LIN {X 0,Y 493.839,Z 352.42,A -85,B 0,C 180,E1 -6409.672,E2 -6409.672} C_VEL
LIN {X 0,Y 494.204,Z 337.139,A -85,B 0,C 180,E1 -6410.171,E2 -6410.171} C_VEL
LIN {X 0,Y 494.44,Z 322.546,A -85,B 0,C 180,E1 -6410.487,E2 -6410.487} C_VEL
LIN {X 0,Y 495.796,Z 177.299,A -85,B 0,C 180,E1 -6412.659,E2 -6412.659} C_VEL
LIN {X 0,Y 492.339,Z 162.269,A -85,B 0,C 180,E1 -6413.065,E2 -6413.065} C_VEL
LIN {X 0,Y 492.169,Z 161.322,A -85,B 0,C 180,E1 -6413.121,E2 -6413.121} C_VEL
LIN {X 0,Y 492.025,Z 155.5,A -85,B 0,C 180,E1 -6413.912,E2 -6413.912} C_VEL
LIN {X 0,Y 488.755,Z 141.231,A -85,B 0,C 180,E1 -6416.241,E2 -6416.241} C_VEL
LIN {X 0,Y 488.72,Z 141.236,A -85,B 0,C 180,E1 -6419.269,E2 -6419.269} C_VEL
LIN {X 0,Y 488.701,Z 141.23,A -85,B 0,C 180,E1 -6422.146,E2 -6422.146} C_VEL
LIN {X 0,Y 488.719,Z 141.234,A -85,B 0,C 180,E1 -6425.113,E2 -6425.113} C_VEL
LIN {X 0,Y 488.676,Z 141.235,A -85,B 0,C 180,E1 -6428.199,E2 -6428.199} C_VEL
LIN {X 0,Y 488.713,Z 141.229,A -85,B 0,C 180,E1 -6431.413,E2 -6431.413} C_VEL
LIN {X 0,Y 488.695,Z 141.23,A -85,B 0,C 180,E1 -6434.023,E2 -6434.023} C_VEL
LIN {X 0,Y 488.702,Z 141.235,A -85,B 0,C 180,E1 -6437.172,E2 -6437.172} C_VEL
LIN {X 0,Y 488.728,Z 141.23,A -85,B 0,C 180,E1 -6439.676,E2 -6439.676} C_VEL
LIN {X 0,Y 488.674,Z 141.234,A -85,B 0,C 180,E1 -6442.276,E2 -6442.276} C_VEL
LIN {X 0,Y 488.72,Z 141.231,A -85,B 0,C 180,E1 -6445.051,E2 -6445.051} C_VEL
LIN {X 0,Y 488.697,Z 141.232,A -85,B 0,C 180,E1 -6448.044,E2 -6448.044} C_VEL
LIN {X 0,Y 488.725,Z 141.225,A -85,B 0,C 180,E1 -6450.73,E2 -6450.73} C_VEL
LIN {X 0,Y 488.747,Z 141.226,A -85,B 0,C 180,E1 -6453.527,E2 -6453.527} C_VEL
LIN {X 0,Y 488.683,Z 141.23,A -85,B 0,C 180,E1 -6456.254,E2 -6456.254} C_VEL
LIN {X 0,Y 488.735,Z 141.229,A -85,B 0,C 180,E1 -6459.175,E2 -6459.175} C_VEL
LIN {X 0,Y 488.748,Z 141.222,A -85,B 0,C 180,E1 -6461.627,E2 -6461.627} C_VEL
LIN {X 0,Y 488.751,Z 141.228,A -85,B 0,C 180,E1 -6464.999,E2 -6464.999} C_VEL
LIN {X 0,Y 488.797,Z 141.216,A -85,B 0,C 180,E1 -6468.387,E2 -6468.387} C_VEL
LIN {X 0,Y 488.807,Z 141.216,A -85,B 0,C 180,E1 -6471.733,E2 -6471.733} C_VEL
LIN {X 0,Y 488.845,Z 141.206,A -85,B 0,C 180,E1 -6474.224,E2 -6474.224} C_VEL
LIN {X 0,Y 488.951,Z 141.2,A -85,B 0,C 180,E1 -6477.528,E2 -6477.528} C_VEL
LIN {X 0,Y 488.957,Z 141.192,A -85,B 0,C 180,E1 -6480,E2 -6480} C_VEL
LIN {X 0,Y 488.951,Z 141.202,A -85,B 0,C 180,E1 -6482.471,E2 -6482.471} C_VEL
LIN {X 0,Y 488.845,Z 141.208,A -85,B 0,C 180,E1 -6485.776,E2 -6485.776} C_VEL
LIN {X 0,Y 488.807,Z 141.215,A -85,B 0,C 180,E1 -6488.266,E2 -6488.266} C_VEL
LIN {X 0,Y 488.797,Z 141.215,A -85,B 0,C 180,E1 -6491.613,E2 -6491.613} C_VEL
LIN {X 0,Y 488.754,Z 141.225,A -85,B 0,C 180,E1 -6495.001,E2 -6495.001} C_VEL
LIN {X 0,Y 488.744,Z 141.224,A -85,B 0,C 180,E1 -6498.442,E2 -6498.442} C_VEL
LIN {X 0,Y 488.702,Z 141.231,A -85,B 0,C 180,E1 -6501.071,E2 -6501.071} C_VEL
LIN {X 0,Y 488.691,Z 141.23,A -85,B 0,C 180,E1 -6503.745,E2 -6503.745} C_VEL
LIN {X 0,Y 488.781,Z 141.222,A -85,B 0,C 180,E1 -6506.944,E2 -6506.944} C_VEL
LIN {X 0,Y 488.7,Z 141.234,A -85,B 0,C 180,E1 -6510.364,E2 -6510.364} C_VEL
LIN {X 0,Y 488.726,Z 141.227,A -85,B 0,C 180,E1 -6513.485,E2 -6513.485} C_VEL
LIN {X 0,Y 488.68,Z 141.24,A -85,B 0,C 180,E1 -6516.357,E2 -6516.357} C_VEL
LIN {X 0,Y 488.692,Z 141.222,A -85,B 0,C 180,E1 -6519.255,E2 -6519.255} C_VEL
LIN {X 0,Y 488.699,Z 141.221,A -85,B 0,C 180,E1 -6521.601,E2 -6521.601} C_VEL
LIN {X 0,Y 488.704,Z 141.232,A -85,B 0,C 180,E1 -6524.802,E2 -6524.802} C_VEL
LIN {X 0,Y 488.724,Z 141.231,A -85,B 0,C 180,E1 -6527.48,E2 -6527.48} C_VEL
LIN {X 0,Y 488.735,Z 141.227,A -85,B 0,C 180,E1 -6530.751,E2 -6530.751} C_VEL
LIN {X 0,Y 488.678,Z 141.236,A -85,B 0,C 180,E1 -6533.87,E2 -6533.87} C_VEL
LIN {X 0,Y 488.735,Z 141.227,A -85,B 0,C 180,E1 -6536.879,E2 -6536.879} C_VEL
LIN {X 0,Y 488.748,Z 141.374,A -85,B 0,C 180,E1 -6537.233,E2 -6537.233} C_VEL
LIN {X 0,Y 495.388,Z 163.433,A -85,B 0,C 180,E1 -6539.928,E2 -6539.928} C_VEL
LIN {X 0,Y 495.755,Z 164.949,A -85,B 0,C 180,E1 -6540.104,E2 -6540.104} C_VEL
LIN {X 0,Y 494.13,Z 196.323,A -85,B 0,C 180,E1 -6543.157,E2 -6543.157} C_VEL
LIN {X 0,Y 492.556,Z 230.849,A -85,B 0,C 180,E1 -6546.453,E2 -6546.453} C_VEL
LIN {X 0,Y 492.243,Z 239.271,A -85,B 0,C 180,E1 -6547.244,E2 -6547.244} C_VEL
LIN {X 0,Y 494.608,Z 258.487,A -85,B 0,C 180,E1 -6547.65,E2 -6547.65} C_VEL
LIN {X 0,Y 493.264,Z 406.875,A -85,B 0,C 180,E1 -6549.87,E2 -6549.87} C_VEL
LIN {X 0,Y 492.832,Z 422.965,A -85,B 0,C 180,E1 -6550.289,E2 -6550.289} C_VEL
LIN {X 0,Y 492.291,Z 437.461,A -85,B 0,C 180,E1 -6550.833,E2 -6550.833} C_VEL
LIN {X 0,Y 491.618,Z 452.169,A -85,B 0,C 180,E1 -6551.563,E2 -6551.563} C_VEL
LIN {X 0,Y 491.046,Z 465.568,A -85,B 0,C 180,E1 -6552.403,E2 -6552.403} C_VEL
LIN {X 0,Y 490.347,Z 479.102,A -85,B 0,C 180,E1 -6553.443,E2 -6553.443} C_VEL
LIN {X 0,Y 489.704,Z 491.563,A -85,B 0,C 180,E1 -6554.604,E2 -6554.604} C_VEL
LIN {X 0,Y 489.214,Z 502.858,A -85,B 0,C 180,E1 -6555.865,E2 -6555.865} C_VEL
LIN {X 0,Y 488.795,Z 513.821,A -85,B 0,C 180,E1 -6557.335,E2 -6557.335} C_VEL
LIN {X 0,Y 488.506,Z 522.941,A -85,B 0,C 180,E1 -6558.802,E2 -6558.802} C_VEL
LIN {X 0,Y 488.294,Z 529.488,A -85,B 0,C 180,E1 -6560.055,E2 -6560.055} C_VEL
LIN {X 0,Y 488.187,Z 536.746,A -85,B 0,C 180,E1 -6561.724,E2 -6561.724} C_VEL
LIN {X 0,Y 488.144,Z 542.565,A -85,B 0,C 180,E1 -6563.423,E2 -6563.423} C_VEL
LIN {X 0,Y 488.156,Z 546.768,A -85,B 0,C 180,E1 -6565.046,E2 -6565.046} C_VEL
LIN {X 0,Y 488.147,Z 549.786,A -85,B 0,C 180,E1 -6566.7,E2 -6566.7} C_VEL
LIN {X 0,Y 488.087,Z 551.58,A -85,B 0,C 180,E1 -6568.351,E2 -6568.351} C_VEL
LIN {X 0,Y 488.175,Z 552.203,A -85,B 0,C 180,E1 -6570.001,E2 -6570.001} C_VEL
LIN {X 0,Y 488.087,Z 551.582,A -85,B 0,C 180,E1 -6571.651,E2 -6571.651} C_VEL
LIN {X 0,Y 488.161,Z 549.786,A -85,B 0,C 180,E1 -6573.302,E2 -6573.302} C_VEL
LIN {X 0,Y 488.157,Z 546.761,A -85,B 0,C 180,E1 -6574.957,E2 -6574.957} C_VEL
LIN {X 0,Y 488.181,Z 542.448,A -85,B 0,C 180,E1 -6576.614,E2 -6576.614} C_VEL
LIN {X 0,Y 488.223,Z 536.742,A -85,B 0,C 180,E1 -6578.278,E2 -6578.278} C_VEL
LIN {X 0,Y 488.322,Z 529.487,A -85,B 0,C 180,E1 -6579.946,E2 -6579.946} C_VEL
LIN {X 0,Y 488.558,Z 521.718,A -85,B 0,C 180,E1 -6581.409,E2 -6581.409} C_VEL
LIN {X 0,Y 488.825,Z 512.358,A -85,B 0,C 180,E1 -6582.877,E2 -6582.877} C_VEL
LIN {X 0,Y 489.235,Z 502.845,A -85,B 0,C 180,E1 -6584.136,E2 -6584.136} C_VEL
LIN {X 0,Y 489.81,Z 490.499,A -85,B 0,C 180,E1 -6585.501,E2 -6585.501} C_VEL
LIN {X 0,Y 490.392,Z 477.894,A -85,B 0,C 180,E1 -6586.657,E2 -6586.657} C_VEL
LIN {X 0,Y 491.072,Z 463.955,A -85,B 0,C 180,E1 -6587.706,E2 -6587.706} C_VEL
LIN {X 0,Y 491.719,Z 450.208,A -85,B 0,C 180,E1 -6588.544,E2 -6588.544} C_VEL
LIN {X 0,Y 492.335,Z 436.099,A -85,B 0,C 180,E1 -6589.224,E2 -6589.224} C_VEL
LIN {X 0,Y 492.874,Z 420.693,A -85,B 0,C 180,E1 -6589.78,E2 -6589.78} C_VEL
LIN {X 0,Y 493.349,Z 405.273,A -85,B 0,C 180,E1 -6590.156,E2 -6590.156} C_VEL
LIN {X 0,Y 494.628,Z 258.388,A -85,B 0,C 180,E1 -6592.349,E2 -6592.349} C_VEL
LIN {X 0,Y 492.076,Z 237.905,A -85,B 0,C 180,E1 -6592.794,E2 -6592.794} C_VEL
LIN {X 0,Y 493.396,Z 209.64,A -85,B 0,C 180,E1 -6595.525,E2 -6595.525} C_VEL
LIN {X 0,Y 495.214,Z 180.207,A -85,B 0,C 180,E1 -6598.496,E2 -6598.496} C_VEL
LIN {X 0,Y 496.295,Z 165.349,A -85,B 0,C 180,E1 -6600.069,E2 -6600.069} C_VEL
LIN {X 0,Y 493.186,Z 154.342,A -85,B 0,C 180,E1 -6601.608,E2 -6601.608} C_VEL
LIN {X 0,Y 489.473,Z 143.554,A -85,B 0,C 180,E1 -6603.327,E2 -6603.327} C_VEL
LIN {X 0,Y 488.734,Z 141.236,A -85,B 0,C 180,E1 -6603.717,E2 -6603.717} C_VEL
LIN {X 0,Y 488.676,Z 141.24,A -85,B 0,C 180,E1 -6606.353,E2 -6606.353} C_VEL
LIN {X 0,Y 488.695,Z 141.238,A -85,B 0,C 180,E1 -6609.256,E2 -6609.256} C_VEL
LIN {X 0,Y 488.669,Z 141.242,A -85,B 0,C 180,E1 -6611.595,E2 -6611.595} C_VEL
LIN {X 0,Y 488.698,Z 141.236,A -85,B 0,C 180,E1 -6614.804,E2 -6614.804} C_VEL
LIN {X 0,Y 488.65,Z 141.243,A -85,B 0,C 180,E1 -6617.47,E2 -6617.47} C_VEL
LIN {X 0,Y 488.671,Z 141.24,A -85,B 0,C 180,E1 -6620.743,E2 -6620.743} C_VEL
LIN {X 0,Y 488.647,Z 141.243,A -85,B 0,C 180,E1 -6623.865,E2 -6623.865} C_VEL
LIN {X 0,Y 488.711,Z 141.237,A -85,B 0,C 180,E1 -6626.521,E2 -6626.521} C_VEL
LIN {X 0,Y 488.701,Z 141.237,A -85,B 0,C 180,E1 -6629.779,E2 -6629.779} C_VEL
LIN {X 0,Y 488.699,Z 141.363,A -85,B 0,C 180,E1 -6631.785,E2 -6631.785} C_VEL
LIN {X 0,Y 491.617,Z 151.425,A -85,B 0,C 180,E1 -6634.065,E2 -6634.065} C_VEL
LIN {X 0,Y 493.665,Z 160.512,A -85,B 0,C 180,E1 -6635.961,E2 -6635.961} C_VEL
LIN {X 0,Y 493.212,Z 170.449,A -85,B 0,C 180,E1 -6637.741,E2 -6637.741} C_VEL
LIN {X 0,Y 492.118,Z 188.229,A -85,B 0,C 180,E1 -6640.824,E2 -6640.824} C_VEL
LIN {X 0,Y 491.433,Z 201.487,A -85,B 0,C 180,E1 -6643.08,E2 -6643.08} C_VEL
LIN {X 0,Y 493.64,Z 211.03,A -85,B 0,C 180,E1 -6643.404,E2 -6643.404} C_VEL
LIN {X 0,Y 491.887,Z 296.371,A -85,B 0,C 180,E1 -6645.071,E2 -6645.071} C_VEL
LIN {X 0,Y 491.644,Z 316.581,A -85,B 0,C 180,E1 -6645.487,E2 -6645.487} C_VEL
LIN {X 0,Y 491.43,Z 330.033,A -85,B 0,C 180,E1 -6645.929,E2 -6645.929} C_VEL
LIN {X 0,Y 491.226,Z 342.558,A -85,B 0,C 180,E1 -6646.52,E2 -6646.52} C_VEL
LIN {X 0,Y 490.825,Z 355.247,A -85,B 0,C 180,E1 -6647.301,E2 -6647.301} C_VEL
LIN {X 0,Y 490.517,Z 365.635,A -85,B 0,C 180,E1 -6648.114,E2 -6648.114} C_VEL
LIN {X 0,Y 490.113,Z 375.332,A -85,B 0,C 180,E1 -6649.047,E2 -6649.047} C_VEL
LIN {X 0,Y 489.837,Z 384.168,A -85,B 0,C 180,E1 -6650.086,E2 -6650.086} C_VEL
LIN {X 0,Y 489.493,Z 392.802,A -85,B 0,C 180,E1 -6651.329,E2 -6651.329} C_VEL
LIN {X 0,Y 489.112,Z 399.707,A -85,B 0,C 180,E1 -6652.57,E2 -6652.57} C_VEL
LIN {X 0,Y 488.987,Z 405.167,A -85,B 0,C 180,E1 -6653.812,E2 -6653.812} C_VEL
LIN {X 0,Y 488.774,Z 409.451,A -85,B 0,C 180,E1 -6655.051,E2 -6655.051} C_VEL
LIN {X 0,Y 488.665,Z 411.692,A -85,B 0,C 180,E1 -6655.876,E2 -6655.876} C_VEL
LIN {X 0,Y 488.63,Z 413.494,A -85,B 0,C 180,E1 -6656.702,E2 -6656.702} C_VEL
LIN {X 0,Y 488.561,Z 414.859,A -85,B 0,C 180,E1 -6657.527,E2 -6657.527} C_VEL
LIN {X 0,Y 488.593,Z 415.773,A -85,B 0,C 180,E1 -6658.352,E2 -6658.352} C_VEL
LIN {X 0,Y 488.501,Z 416.452,A -85,B 0,C 180,E1 -6660,E2 -6660} C_VEL
LIN {X 0,Y 488.515,Z 416.169,A -85,B 0,C 180,E1 -6660.824,E2 -6660.824} C_VEL
LIN {X 0,Y 488.442,Z 415.482,A -85,B 0,C 180,E1 -6661.649,E2 -6661.649} C_VEL
LIN {X 0,Y 488.545,Z 414.383,A -85,B 0,C 180,E1 -6662.474,E2 -6662.474} C_VEL
LIN {X 0,Y 488.474,Z 412.907,A -85,B 0,C 180,E1 -6663.299,E2 -6663.299} C_VEL
LIN {X 0,Y 488.647,Z 409.812,A -85,B 0,C 180,E1 -6664.537,E2 -6664.537} C_VEL
LIN {X 0,Y 488.67,Z 405.702,A -85,B 0,C 180,E1 -6665.778,E2 -6665.778} C_VEL
LIN {X 0,Y 488.929,Z 400.458,A -85,B 0,C 180,E1 -6667.009,E2 -6667.009} C_VEL
LIN {X 0,Y 489.141,Z 393.783,A -85,B 0,C 180,E1 -6668.261,E2 -6668.261} C_VEL
LIN {X 0,Y 489.391,Z 385.54,A -85,B 0,C 180,E1 -6669.506,E2 -6669.506} C_VEL
LIN {X 0,Y 489.695,Z 377.139,A -85,B 0,C 180,E1 -6670.544,E2 -6670.544} C_VEL
LIN {X 0,Y 490.004,Z 366.899,A -85,B 0,C 180,E1 -6671.584,E2 -6671.584} C_VEL
LIN {X 0,Y 490.403,Z 355.297,A -85,B 0,C 180,E1 -6672.521,E2 -6672.521} C_VEL
LIN {X 0,Y 490.668,Z 344.057,A -85,B 0,C 180,E1 -6673.249,E2 -6673.249} C_VEL
LIN {X 0,Y 490.938,Z 331.583,A -85,B 0,C 180,E1 -6673.874,E2 -6673.874} C_VEL
LIN {X 0,Y 491.119,Z 319.461,A -85,B 0,C 180,E1 -6674.318,E2 -6674.318} C_VEL
LIN {X 0,Y 491.297,Z 305.308,A -85,B 0,C 180,E1 -6674.656,E2 -6674.656} C_VEL
LIN {X 0,Y 492.302,Z 209.873,A -85,B 0,C 180,E1 -6676.239,E2 -6676.239} C_VEL
LIN {X 0,Y 490.118,Z 198.052,A -85,B 0,C 180,E1 -6676.525,E2 -6676.525} C_VEL
LIN {X 0,Y 490.795,Z 177.36,A -85,B 0,C 180,E1 -6679.883,E2 -6679.883} C_VEL
LIN {X 0,Y 491.408,Z 160.1,A -85,B 0,C 180,E1 -6682.715,E2 -6682.715} C_VEL
LIN {X 0,Y 491.449,Z 153.87,A -85,B 0,C 180,E1 -6683.759,E2 -6683.759} C_VEL
LIN {X 0,Y 488.758,Z 141.23,A -85,B 0,C 180,E1 -6686.07,E2 -6686.07} C_VEL
LIN {X 0,Y 488.714,Z 141.237,A -85,B 0,C 180,E1 -6689.271,E2 -6689.271} C_VEL
LIN {X 0,Y 488.708,Z 141.232,A -85,B 0,C 180,E1 -6692.147,E2 -6692.147} C_VEL
LIN {X 0,Y 488.72,Z 141.235,A -85,B 0,C 180,E1 -6695.115,E2 -6695.115} C_VEL
LIN {X 0,Y 488.681,Z 141.234,A -85,B 0,C 180,E1 -6698.2,E2 -6698.2} C_VEL
LIN {X 0,Y 488.723,Z 141.225,A -85,B 0,C 180,E1 -6700.344,E2 -6700.344} C_VEL
LIN {X 0,Y 488.682,Z 141.233,A -85,B 0,C 180,E1 -6703.655,E2 -6703.655} C_VEL
LIN {X 0,Y 488.689,Z 141.234,A -85,B 0,C 180,E1 -6706.266,E2 -6706.266} C_VEL
LIN {X 0,Y 488.021,Z 141.32,A -85,B 0,C 180,E1 -6706.953,E2 -6706.953} C_VEL
LIN {X 0,Y 485.159,Z 141.675,A -85,B 0,C 180,E1 -6708.07,E2 -6708.07} C_VEL
LIN {X 0,Y 482.754,Z 141.979,A -85,B 0,C 180,E1 -6708.97,E2 -6708.97} C_VEL
LIN {X 0,Y 481.742,Z 142.098,A -85,B 0,C 180,E1 -6709.665,E2 -6709.665} C_VEL
LIN {X 0,Y 481.671,Z 142.105,A -85,B 0,C 180,E1 -6709.9,E2 -6709.9} C_VEL
LIN {X 0,Y 481.634,Z 142.115,A -85,B 0,C 180,E1 -6712.202,E2 -6712.202} C_VEL
LIN {X 0,Y 481.689,Z 142.111,A -85,B 0,C 180,E1 -6715.317,E2 -6715.317} C_VEL
LIN {X 0,Y 481.649,Z 142.116,A -85,B 0,C 180,E1 -6718.311,E2 -6718.311} C_VEL
LIN {X 0,Y 481.702,Z 142.108,A -85,B 0,C 180,E1 -6721.218,E2 -6721.218} C_VEL
LIN {X 0,Y 481.759,Z 142.217,A -85,B 0,C 180,E1 -6723.58,E2 -6723.58} C_VEL
LIN {X 0,Y 484.847,Z 155.51,A -85,B 0,C 180,E1 -6725.744,E2 -6725.744} C_VEL
LIN {X 0,Y 485.468,Z 161.01,A -85,B 0,C 180,E1 -6726.538,E2 -6726.538} C_VEL
LIN {X 0,Y 485.507,Z 162.139,A -85,B 0,C 180,E1 -6726.674,E2 -6726.674} C_VEL
LIN {X 0,Y 489.208,Z 177.555,A -85,B 0,C 180,E1 -6727.108,E2 -6727.108} C_VEL
LIN {X 0,Y 488.095,Z 293.925,A -85,B 0,C 180,E1 -6728.873,E2 -6728.873} C_VEL
LIN {X 0,Y 487.695,Z 329.765,A -85,B 0,C 180,E1 -6729.443,E2 -6729.443} C_VEL
LIN {X 0,Y 487.382,Z 345.225,A -85,B 0,C 180,E1 -6729.862,E2 -6729.862} C_VEL
LIN {X 0,Y 486.934,Z 360.24,A -85,B 0,C 180,E1 -6730.447,E2 -6730.447} C_VEL
LIN {X 0,Y 486.448,Z 373.705,A -85,B 0,C 180,E1 -6731.139,E2 -6731.139} C_VEL
LIN {X 0,Y 485.777,Z 386.96,A -85,B 0,C 180,E1 -6731.985,E2 -6731.985} C_VEL
LIN {X 0,Y 485.114,Z 398.493,A -85,B 0,C 180,E1 -6732.88,E2 -6732.88} C_VEL
LIN {X 0,Y 484.405,Z 410.523,A -85,B 0,C 180,E1 -6733.998,E2 -6733.998} C_VEL
LIN {X 0,Y 483.672,Z 421.927,A -85,B 0,C 180,E1 -6735.268,E2 -6735.268} C_VEL
LIN {X 0,Y 483.039,Z 431.517,A -85,B 0,C 180,E1 -6736.538,E2 -6736.538} C_VEL
LIN {X 0,Y 482.468,Z 441.015,A -85,B 0,C 180,E1 -6738.043,E2 -6738.043} C_VEL
LIN {X 0,Y 482.005,Z 448.674,A -85,B 0,C 180,E1 -6739.498,E2 -6739.498} C_VEL
LIN {X 0,Y 481.645,Z 455.916,A -85,B 0,C 180,E1 -6741.186,E2 -6741.186} C_VEL
LIN {X 0,Y 481.353,Z 461.78,A -85,B 0,C 180,E1 -6742.912,E2 -6742.912} C_VEL
LIN {X 0,Y 481.162,Z 465.052,A -85,B 0,C 180,E1 -6744.131,E2 -6744.131} C_VEL
LIN {X 0,Y 481.116,Z 468.502,A -85,B 0,C 180,E1 -6745.81,E2 -6745.81} C_VEL
LIN {X 0,Y 480.955,Z 470.792,A -85,B 0,C 180,E1 -6747.486,E2 -6747.486} C_VEL
LIN {X 0,Y 480.84,Z 471.96,A -85,B 0,C 180,E1 -6749.161,E2 -6749.161} C_VEL
LIN {X 0,Y 480.839,Z 471.977,A -85,B 0,C 180,E1 -6750.836,E2 -6750.836} C_VEL
LIN {X 0,Y 480.954,Z 470.872,A -85,B 0,C 180,E1 -6752.511,E2 -6752.511} C_VEL
LIN {X 0,Y 481.105,Z 468.653,A -85,B 0,C 180,E1 -6754.188,E2 -6754.188} C_VEL
LIN {X 0,Y 481.153,Z 465.28,A -85,B 0,C 180,E1 -6755.867,E2 -6755.867} C_VEL
LIN {X 0,Y 481.397,Z 460.64,A -85,B 0,C 180,E1 -6757.549,E2 -6757.549} C_VEL
LIN {X 0,Y 481.696,Z 454.617,A -85,B 0,C 180,E1 -6759.234,E2 -6759.234} C_VEL
LIN {X 0,Y 482.097,Z 447.036,A -85,B 0,C 180,E1 -6760.923,E2 -6760.923} C_VEL
LIN {X 0,Y 482.586,Z 438.585,A -85,B 0,C 180,E1 -6762.462,E2 -6762.462} C_VEL
LIN {X 0,Y 483.218,Z 429.172,A -85,B 0,C 180,E1 -6763.884,E2 -6763.884} C_VEL
LIN {X 0,Y 483.854,Z 419.185,A -85,B 0,C 180,E1 -6765.155,E2 -6765.155} C_VEL
LIN {X 0,Y 484.57,Z 407.686,A -85,B 0,C 180,E1 -6766.382,E2 -6766.382} C_VEL
LIN {X 0,Y 485.297,Z 395.497,A -85,B 0,C 180,E1 -6767.465,E2 -6767.465} C_VEL
LIN {X 0,Y 486.024,Z 382.137,A -85,B 0,C 180,E1 -6768.439,E2 -6768.439} C_VEL
LIN {X 0,Y 486.644,Z 367.616,A -85,B 0,C 180,E1 -6769.289,E2 -6769.289} C_VEL
LIN {X 0,Y 487.186,Z 353.095,A -85,B 0,C 180,E1 -6769.946,E2 -6769.946} C_VEL
LIN {X 0,Y 487.567,Z 338.673,A -85,B 0,C 180,E1 -6770.431,E2 -6770.431} C_VEL
LIN {X 0,Y 487.809,Z 322.974,A -85,B 0,C 180,E1 -6770.778,E2 -6770.778} C_VEL
LIN {X 0,Y 489.274,Z 178.987,A -85,B 0,C 180,E1 -6772.958,E2 -6772.958} C_VEL
LIN {X 0,Y 488.771,Z 175.625,A -85,B 0,C 180,E1 -6773.037,E2 -6773.037} C_VEL
LIN {X 0,Y 485.465,Z 161.934,A -85,B 0,C 180,E1 -6773.44,E2 -6773.44} C_VEL
LIN {X 0,Y 485.159,Z 156.905,A -85,B 0,C 180,E1 -6774.13,E2 -6774.13} C_VEL
LIN {X 0,Y 481.862,Z 142.831,A -85,B 0,C 180,E1 -6776.412,E2 -6776.412} C_VEL
LIN {X 0,Y 481.72,Z 142.107,A -85,B 0,C 180,E1 -6776.537,E2 -6776.537} C_VEL
LIN {X 0,Y 481.675,Z 142.113,A -85,B 0,C 180,E1 -6779.74,E2 -6779.74} C_VEL
LIN {X 0,Y 481.669,Z 142.106,A -85,B 0,C 180,E1 -6782.673,E2 -6782.673} C_VEL
LIN {X 0,Y 481.638,Z 142.117,A -85,B 0,C 180,E1 -6785.708,E2 -6785.708} C_VEL
LIN {X 0,Y 481.666,Z 142.11,A -85,B 0,C 180,E1 -6788.858,E2 -6788.858} C_VEL
LIN {X 0,Y 481.656,Z 142.111,A -85,B 0,C 180,E1 -6791.913,E2 -6791.913} C_VEL
LIN {X 0,Y 481.653,Z 142.106,A -85,B 0,C 180,E1 -6794.456,E2 -6794.456} C_VEL
LIN {X 0,Y 481.641,Z 142.111,A -85,B 0,C 180,E1 -6797.838,E2 -6797.838} C_VEL
LIN {X 0,Y 481.712,Z 142.103,A -85,B 0,C 180,E1 -6800.644,E2 -6800.644} C_VEL
LIN {X 0,Y 481.634,Z 142.111,A -85,B 0,C 180,E1 -6804.29,E2 -6804.29} C_VEL
LIN {X 0,Y 481.664,Z 142.114,A -85,B 0,C 180,E1 -6807.325,E2 -6807.325} C_VEL
LIN {X 0,Y 481.679,Z 142.098,A -85,B 0,C 180,E1 -6810.259,E2 -6810.259} C_VEL
LIN {X 0,Y 481.736,Z 142.105,A -85,B 0,C 180,E1 -6813.111,E2 -6813.111} C_VEL
LIN {X 0,Y 481.667,Z 142.103,A -85,B 0,C 180,E1 -6815.886,E2 -6815.886} C_VEL
LIN {X 0,Y 481.692,Z 142.108,A -85,B 0,C 180,E1 -6819.027,E2 -6819.027} C_VEL
LIN {X 0,Y 481.697,Z 142.1,A -85,B 0,C 180,E1 -6822.158,E2 -6822.158} C_VEL
LIN {X 0,Y 481.731,Z 142.106,A -85,B 0,C 180,E1 -6824.775,E2 -6824.775} C_VEL
LIN {X 0,Y 481.742,Z 142.093,A -85,B 0,C 180,E1 -6828.215,E2 -6828.215} C_VEL
LIN {X 0,Y 481.752,Z 142.095,A -85,B 0,C 180,E1 -6831.611,E2 -6831.611} C_VEL
LIN {X 0,Y 481.806,Z 142.082,A -85,B 0,C 180,E1 -6834.139,E2 -6834.139} C_VEL
LIN {X 0,Y 481.918,Z 142.076,A -85,B 0,C 180,E1 -6837.492,E2 -6837.492} C_VEL
LIN {X 0,Y 481.928,Z 142.067,A -85,B 0,C 180,E1 -6840,E2 -6840} C_VEL
LIN {X 0,Y 481.918,Z 142.078,A -85,B 0,C 180,E1 -6842.507,E2 -6842.507} C_VEL
LIN {X 0,Y 481.806,Z 142.085,A -85,B 0,C 180,E1 -6845.86,E2 -6845.86} C_VEL
LIN {X 0,Y 481.753,Z 142.095,A -85,B 0,C 180,E1 -6848.388,E2 -6848.388} C_VEL
LIN {X 0,Y 481.741,Z 142.094,A -85,B 0,C 180,E1 -6851.785,E2 -6851.785} C_VEL
LIN {X 0,Y 481.733,Z 142.098,A -85,B 0,C 180,E1 -6855.224,E2 -6855.224} C_VEL
LIN {X 0,Y 481.701,Z 142.098,A -85,B 0,C 180,E1 -6858.722,E2 -6858.722} C_VEL
LIN {X 0,Y 481.643,Z 142.109,A -85,B 0,C 180,E1 -6861.395,E2 -6861.395} C_VEL
LIN {X 0,Y 481.672,Z 142.107,A -85,B 0,C 180,E1 -6864.113,E2 -6864.113} C_VEL
LIN {X 0,Y 481.736,Z 142.099,A -85,B 0,C 180,E1 -6867.14,E2 -6867.14} C_VEL
LIN {X 0,Y 481.668,Z 142.103,A -85,B 0,C 180,E1 -6869.742,E2 -6869.742} C_VEL
LIN {X 0,Y 481.663,Z 142.109,A -85,B 0,C 180,E1 -6872.675,E2 -6872.675} C_VEL
LIN {X 0,Y 481.634,Z 142.112,A -85,B 0,C 180,E1 -6875.71,E2 -6875.71} C_VEL
LIN {X 0,Y 481.662,Z 142.098,A -85,B 0,C 180,E1 -6878.86,E2 -6878.86} C_VEL
LIN {X 0,Y 481.644,Z 142.103,A -85,B 0,C 180,E1 -6881.914,E2 -6881.914} C_VEL
LIN {X 0,Y 481.651,Z 142.114,A -85,B 0,C 180,E1 -6884.458,E2 -6884.458} C_VEL
LIN {X 0,Y 481.681,Z 142.107,A -85,B 0,C 180,E1 -6886.847,E2 -6886.847} C_VEL
LIN {X 0,Y 481.682,Z 142.112,A -85,B 0,C 180,E1 -6890.062,E2 -6890.062} C_VEL
LIN {X 0,Y 481.622,Z 142.112,A -85,B 0,C 180,E1 -6893.254,E2 -6893.254} C_VEL
LIN {X 0,Y 481.704,Z 142.104,A -85,B 0,C 180,E1 -6896.331,E2 -6896.331} C_VEL
LIN {X 0,Y 481.704,Z 142.197,A -85,B 0,C 180,E1 -6896.864,E2 -6896.864} C_VEL
LIN {X 0,Y 488.523,Z 164.814,A -85,B 0,C 180,E1 -6899.675,E2 -6899.675} C_VEL
LIN {X 0,Y 489.019,Z 168.078,A -85,B 0,C 180,E1 -6900.04,E2 -6900.04} C_VEL
LIN {X 0,Y 487.185,Z 201.325,A -85,B 0,C 180,E1 -6903.322,E2 -6903.322} C_VEL
LIN {X 0,Y 485.575,Z 234.709,A -85,B 0,C 180,E1 -6906.547,E2 -6906.547} C_VEL
LIN {X 0,Y 485.399,Z 238.384,A -85,B 0,C 180,E1 -6906.898,E2 -6906.898} C_VEL
LIN {X 0,Y 488.023,Z 259.965,A -85,B 0,C 180,E1 -6907.362,E2 -6907.362} C_VEL
LIN {X 0,Y 486.598,Z 406.396,A -85,B 0,C 180,E1 -6909.582,E2 -6909.582} C_VEL
LIN {X 0,Y 486.128,Z 422.117,A -85,B 0,C 180,E1 -6909.995,E2 -6909.995} C_VEL
LIN {X 0,Y 485.544,Z 436.913,A -85,B 0,C 180,E1 -6910.556,E2 -6910.556} C_VEL
LIN {X 0,Y 484.854,Z 451.61,A -85,B 0,C 180,E1 -6911.296,E2 -6911.296} C_VEL
LIN {X 0,Y 484.199,Z 464.998,A -85,B 0,C 180,E1 -6912.145,E2 -6912.145} C_VEL
LIN {X 0,Y 483.414,Z 478.664,A -85,B 0,C 180,E1 -6913.211,E2 -6913.211} C_VEL
LIN {X 0,Y 482.777,Z 490.983,A -85,B 0,C 180,E1 -6914.378,E2 -6914.378} C_VEL
LIN {X 0,Y 482.2,Z 502.272,A -85,B 0,C 180,E1 -6915.655,E2 -6915.655} C_VEL
LIN {X 0,Y 481.767,Z 513.235,A -85,B 0,C 180,E1 -6917.147,E2 -6917.147} C_VEL
LIN {X 0,Y 481.422,Z 522.351,A -85,B 0,C 180,E1 -6918.635,E2 -6918.635} C_VEL
LIN {X 0,Y 481.247,Z 528.902,A -85,B 0,C 180,E1 -6919.908,E2 -6919.908} C_VEL
LIN {X 0,Y 481.096,Z 536.158,A -85,B 0,C 180,E1 -6921.601,E2 -6921.601} C_VEL
LIN {X 0,Y 481.069,Z 542.271,A -85,B 0,C 180,E1 -6923.423,E2 -6923.423} C_VEL
LIN {X 0,Y 481.069,Z 546.177,A -85,B 0,C 180,E1 -6924.972,E2 -6924.972} C_VEL
LIN {X 0,Y 481.067,Z 549.197,A -85,B 0,C 180,E1 -6926.651,E2 -6926.651} C_VEL
LIN {X 0,Y 481.009,Z 550.995,A -85,B 0,C 180,E1 -6928.327,E2 -6928.327} C_VEL
LIN {X 0,Y 481.1,Z 551.618,A -85,B 0,C 180,E1 -6930.001,E2 -6930.001} C_VEL
LIN {X 0,Y 481.009,Z 550.997,A -85,B 0,C 180,E1 -6931.676,E2 -6931.676} C_VEL
LIN {X 0,Y 481.079,Z 549.201,A -85,B 0,C 180,E1 -6933.351,E2 -6933.351} C_VEL
LIN {X 0,Y 481.068,Z 546.175,A -85,B 0,C 180,E1 -6935.03,E2 -6935.03} C_VEL
LIN {X 0,Y 481.09,Z 541.86,A -85,B 0,C 180,E1 -6936.712,E2 -6936.712} C_VEL
LIN {X 0,Y 481.127,Z 536.153,A -85,B 0,C 180,E1 -6938.4,E2 -6938.4} C_VEL
LIN {X 0,Y 481.276,Z 528.902,A -85,B 0,C 180,E1 -6940.093,E2 -6940.093} C_VEL
LIN {X 0,Y 481.477,Z 521.128,A -85,B 0,C 180,E1 -6941.579,E2 -6941.579} C_VEL
LIN {X 0,Y 481.796,Z 511.769,A -85,B 0,C 180,E1 -6943.069,E2 -6943.069} C_VEL
LIN {X 0,Y 482.226,Z 502.256,A -85,B 0,C 180,E1 -6944.346,E2 -6944.346} C_VEL
LIN {X 0,Y 482.805,Z 490.958,A -85,B 0,C 180,E1 -6945.623,E2 -6945.623} C_VEL
LIN {X 0,Y 483.421,Z 478.624,A -85,B 0,C 180,E1 -6946.791,E2 -6946.791} C_VEL
LIN {X 0,Y 484.152,Z 464.958,A -85,B 0,C 180,E1 -6947.859,E2 -6947.859} C_VEL
LIN {X 0,Y 484.854,Z 451.57,A -85,B 0,C 180,E1 -6948.706,E2 -6948.706} C_VEL
LIN {X 0,Y 485.553,Z 436.839,A -85,B 0,C 180,E1 -6949.446,E2 -6949.446} C_VEL
LIN {X 0,Y 486.159,Z 421.046,A -85,B 0,C 180,E1 -6950.038,E2 -6950.038} C_VEL
LIN {X 0,Y 486.635,Z 406.241,A -85,B 0,C 180,E1 -6950.419,E2 -6950.419} C_VEL
LIN {X 0,Y 487.983,Z 265.524,A -85,B 0,C 180,E1 -6952.552,E2 -6952.552} C_VEL
LIN {X 0,Y 487.853,Z 257.529,A -85,B 0,C 180,E1 -6952.683,E2 -6952.683} C_VEL
LIN {X 0,Y 485.321,Z 237.456,A -85,B 0,C 180,E1 -6953.13,E2 -6953.13} C_VEL
LIN {X 0,Y 486.832,Z 208.642,A -85,B 0,C 180,E1 -6955.98,E2 -6955.98} C_VEL
LIN {X 0,Y 488.923,Z 179.066,A -85,B 0,C 180,E1 -6959.054,E2 -6959.054} C_VEL
LIN {X 0,Y 489.807,Z 167.522,A -85,B 0,C 180,E1 -6960.313,E2 -6960.313} C_VEL
LIN {X 0,Y 486.441,Z 155.904,A -85,B 0,C 180,E1 -6962.014,E2 -6962.014} C_VEL
LIN {X 0,Y 483.251,Z 146.677,A -85,B 0,C 180,E1 -6963.549,E2 -6963.549} C_VEL
LIN {X 0,Y 481.689,Z 142.113,A -85,B 0,C 180,E1 -6964.397,E2 -6964.397} C_VEL
LIN {X 0,Y 481.651,Z 142.116,A -85,B 0,C 180,E1 -6968.007,E2 -6968.007} C_VEL
LIN {X 0,Y 481.625,Z 142.118,A -85,B 0,C 180,E1 -6971.046,E2 -6971.046} C_VEL
LIN {X 0,Y 481.652,Z 142.113,A -85,B 0,C 180,E1 -6974.459,E2 -6974.459} C_VEL
LIN {X 0,Y 481.615,Z 142.119,A -85,B 0,C 180,E1 -6976.856,E2 -6976.856} C_VEL
LIN {X 0,Y 481.63,Z 142.116,A -85,B 0,C 180,E1 -6980.055,E2 -6980.055} C_VEL
LIN {X 0,Y 481.607,Z 142.122,A -85,B 0,C 180,E1 -6983.251,E2 -6983.251} C_VEL
LIN {X 0,Y 481.674,Z 142.113,A -85,B 0,C 180,E1 -6986.327,E2 -6986.327} C_VEL
LIN {X 0,Y 481.63,Z 142.119,A -85,B 0,C 180,E1 -6989.423,E2 -6989.423} C_VEL
LIN {X 0,Y 481.639,Z 142.121,A -85,B 0,C 180,E1 -6991.107,E2 -6991.107} C_VEL
LIN {X 0,Y 484.637,Z 152.205,A -85,B 0,C 180,E1 -6993.501,E2 -6993.501} C_VEL
LIN {X 0,Y 486.991,Z 162.378,A -85,B 0,C 180,E1 -6995.701,E2 -6995.701} C_VEL
LIN {X 0,Y 486.951,Z 167.235,A -85,B 0,C 180,E1 -6996.616,E2 -6996.616} C_VEL
LIN {X 0,Y 485.774,Z 184.506,A -85,B 0,C 180,E1 -6999.683,E2 -6999.683} C_VEL
LIN {X 0,Y 484.737,Z 202.088,A -85,B 0,C 180,E1 -7002.731,E2 -7002.731} C_VEL
LIN {X 0,Y 487.157,Z 213.037,A -85,B 0,C 180,E1 -7003.111,E2 -7003.111} C_VEL
LIN {X 0,Y 485.068,Z 303.409,A -85,B 0,C 180,E1 -7004.937,E2 -7004.937} C_VEL
LIN {X 0,Y 484.878,Z 319.654,A -85,B 0,C 180,E1 -7005.306,E2 -7005.306} C_VEL
LIN {X 0,Y 484.661,Z 332.854,A -85,B 0,C 180,E1 -7005.782,E2 -7005.782} C_VEL
LIN {X 0,Y 484.388,Z 345.921,A -85,B 0,C 180,E1 -7006.437,E2 -7006.437} C_VEL
LIN {X 0,Y 483.977,Z 357.501,A -85,B 0,C 180,E1 -7007.19,E2 -7007.19} C_VEL
LIN {X 0,Y 483.63,Z 367.977,A -85,B 0,C 180,E1 -7008.049,E2 -7008.049} C_VEL
LIN {X 0,Y 483.23,Z 378.404,A -85,B 0,C 180,E1 -7009.102,E2 -7009.102} C_VEL
LIN {X 0,Y 482.896,Z 386.905,A -85,B 0,C 180,E1 -7010.154,E2 -7010.154} C_VEL
LIN {X 0,Y 482.471,Z 395.166,A -85,B 0,C 180,E1 -7011.413,E2 -7011.413} C_VEL
LIN {X 0,Y 482.176,Z 402.011,A -85,B 0,C 180,E1 -7012.723,E2 -7012.723} C_VEL
LIN {X 0,Y 481.918,Z 407.83,A -85,B 0,C 180,E1 -7014.141,E2 -7014.141} C_VEL
LIN {X 0,Y 481.763,Z 411.722,A -85,B 0,C 180,E1 -7015.398,E2 -7015.398} C_VEL
LIN {X 0,Y 481.637,Z 414.556,A -85,B 0,C 180,E1 -7016.654,E2 -7016.654} C_VEL
LIN {X 0,Y 481.548,Z 415.909,A -85,B 0,C 180,E1 -7017.491,E2 -7017.491} C_VEL
LIN {X 0,Y 481.579,Z 416.809,A -85,B 0,C 180,E1 -7018.328,E2 -7018.328} C_VEL
LIN {X 0,Y 481.509,Z 417.333,A -85,B 0,C 180,E1 -7019.164,E2 -7019.164} C_VEL
LIN {X 0,Y 481.481,Z 417.46,A -85,B 0,C 180,E1 -7020,E2 -7020} C_VEL
LIN {X 0,Y 481.496,Z 417.157,A -85,B 0,C 180,E1 -7020.836,E2 -7020.836} C_VEL
LIN {X 0,Y 481.419,Z 416.45,A -85,B 0,C 180,E1 -7021.673,E2 -7021.673} C_VEL
LIN {X 0,Y 481.527,Z 415.329,A -85,B 0,C 180,E1 -7022.51,E2 -7022.51} C_VEL
LIN {X 0,Y 481.446,Z 413.835,A -85,B 0,C 180,E1 -7023.348,E2 -7023.348} C_VEL
LIN {X 0,Y 481.631,Z 410.7,A -85,B 0,C 180,E1 -7024.603,E2 -7024.603} C_VEL
LIN {X 0,Y 481.672,Z 406.546,A -85,B 0,C 180,E1 -7025.862,E2 -7025.862} C_VEL
LIN {X 0,Y 481.942,Z 401.308,A -85,B 0,C 180,E1 -7027.099,E2 -7027.099} C_VEL
LIN {X 0,Y 482.17,Z 394.518,A -85,B 0,C 180,E1 -7028.381,E2 -7028.381} C_VEL
LIN {X 0,Y 482.425,Z 386.211,A -85,B 0,C 180,E1 -7029.644,E2 -7029.644} C_VEL
LIN {X 0,Y 482.753,Z 377.746,A -85,B 0,C 180,E1 -7030.697,E2 -7030.697} C_VEL
LIN {X 0,Y 483.082,Z 367.426,A -85,B 0,C 180,E1 -7031.752,E2 -7031.752} C_VEL
LIN {X 0,Y 483.498,Z 355.851,A -85,B 0,C 180,E1 -7032.695,E2 -7032.695} C_VEL
LIN {X 0,Y 483.765,Z 344.416,A -85,B 0,C 180,E1 -7033.441,E2 -7033.441} C_VEL
LIN {X 0,Y 484.059,Z 331.791,A -85,B 0,C 180,E1 -7034.075,E2 -7034.075} C_VEL
LIN {X 0,Y 484.236,Z 318.63,A -85,B 0,C 180,E1 -7034.553,E2 -7034.553} C_VEL
LIN {X 0,Y 484.43,Z 305.125,A -85,B 0,C 180,E1 -7034.869,E2 -7034.869} C_VEL
LIN {X 0,Y 485.49,Z 210.169,A -85,B 0,C 180,E1 -7036.48,E2 -7036.48} C_VEL
LIN {X 0,Y 483.221,Z 198.271,A -85,B 0,C 180,E1 -7036.783,E2 -7036.783} C_VEL
LIN {X 0,Y 483.937,Z 177.559,A -85,B 0,C 180,E1 -7040.176,E2 -7040.176} C_VEL
LIN {X 0,Y 484.649,Z 158.877,A -85,B 0,C 180,E1 -7043.276,E2 -7043.276} C_VEL
LIN {X 0,Y 484.465,Z 154.899,A -85,B 0,C 180,E1 -7043.966,E2 -7043.966} C_VEL
LIN {X 0,Y 481.701,Z 142.109,A -85,B 0,C 180,E1 -7046.306,E2 -7046.306} C_VEL
LIN {X 0,Y 481.677,Z 142.113,A -85,B 0,C 180,E1 -7049.741,E2 -7049.741} C_VEL
LIN {X 0,Y 481.677,Z 142.108,A -85,B 0,C 180,E1 -7052.674,E2 -7052.674} C_VEL
LIN {X 0,Y 481.637,Z 142.115,A -85,B 0,C 180,E1 -7055.71,E2 -7055.71} C_VEL
LIN {X 0,Y 481.673,Z 142.111,A -85,B 0,C 180,E1 -7058.859,E2 -7058.859} C_VEL
LIN {X 0,Y 481.65,Z 142.111,A -85,B 0,C 180,E1 -7061.911,E2 -7061.911} C_VEL
LIN {X 0,Y 481.659,Z 142.107,A -85,B 0,C 180,E1 -7064.458,E2 -7064.458} C_VEL
LIN {X 0,Y 481.652,Z 142.111,A -85,B 0,C 180,E1 -7067.839,E2 -7067.839} C_VEL
LIN {X 0,Y 481.671,Z 142.105,A -85,B 0,C 180,E1 -7069.9,E2 -7069.9} C_VEL
LIN {X 0,Y 481.021,Z 142.192,A -85,B 0,C 180,E1 -7070.598,E2 -7070.598} C_VEL
LIN {X 0,Y 478.13,Z 142.551,A -85,B 0,C 180,E1 -7071.73,E2 -7071.73} C_VEL
LIN {X 0,Y 475.685,Z 142.858,A -85,B 0,C 180,E1 -7072.642,E2 -7072.642} C_VEL
LIN {X 0,Y 474.658,Z 142.987,A -85,B 0,C 180,E1 -7073.348,E2 -7073.348} C_VEL
LIN {X 0,Y 474.587,Z 142.994,A -85,B 0,C 180,E1 -7073.587,E2 -7073.587} C_VEL
LIN {X 0,Y 474.629,Z 142.99,A -85,B 0,C 180,E1 -7076.778,E2 -7076.778} C_VEL
LIN {X 0,Y 474.608,Z 142.99,A -85,B 0,C 180,E1 -7079.769,E2 -7079.769} C_VEL
LIN {X 0,Y 474.731,Z 142.978,A -85,B 0,C 180,E1 -7083.246,E2 -7083.246} C_VEL
LIN {X 0,Y 478.199,Z 157.937,A -85,B 0,C 180,E1 -7085.672,E2 -7085.672} C_VEL
LIN {X 0,Y 478.802,Z 162.707,A -85,B 0,C 180,E1 -7086.328,E2 -7086.328} C_VEL
LIN {X 0,Y 482.748,Z 179.203,A -85,B 0,C 180,E1 -7086.802,E2 -7086.802} C_VEL
LIN {X 0,Y 481.24,Z 317.706,A -85,B 0,C 180,E1 -7088.925,E2 -7088.925} C_VEL
LIN {X 0,Y 481.001,Z 334.574,A -85,B 0,C 180,E1 -7089.247,E2 -7089.247} C_VEL
LIN {X 0,Y 480.645,Z 349.71,A -85,B 0,C 180,E1 -7089.711,E2 -7089.711} C_VEL
LIN {X 0,Y 480.162,Z 364.183,A -85,B 0,C 180,E1 -7090.326,E2 -7090.326} C_VEL
LIN {X 0,Y 479.574,Z 377.875,A -85,B 0,C 180,E1 -7091.08,E2 -7091.08} C_VEL
LIN {X 0,Y 478.873,Z 390.5,A -85,B 0,C 180,E1 -7091.938,E2 -7091.938} C_VEL
LIN {X 0,Y 477.994,Z 403.874,A -85,B 0,C 180,E1 -7093.053,E2 -7093.053} C_VEL
LIN {X 0,Y 477.343,Z 415.178,A -85,B 0,C 180,E1 -7094.193,E2 -7094.193} C_VEL
LIN {X 0,Y 476.623,Z 425.926,A -85,B 0,C 180,E1 -7095.482,E2 -7095.482} C_VEL
LIN {X 0,Y 475.935,Z 435.254,A -85,B 0,C 180,E1 -7096.811,E2 -7096.811} C_VEL
LIN {X 0,Y 475.385,Z 443.84,A -85,B 0,C 180,E1 -7098.27,E2 -7098.27} C_VEL
LIN {X 0,Y 474.9,Z 451.202,A -85,B 0,C 180,E1 -7099.77,E2 -7099.77} C_VEL
LIN {X 0,Y 474.527,Z 458.056,A -85,B 0,C 180,E1 -7101.482,E2 -7101.482} C_VEL
LIN {X 0,Y 474.262,Z 463.441,A -85,B 0,C 180,E1 -7103.191,E2 -7103.191} C_VEL
LIN {X 0,Y 474.125,Z 467.51,A -85,B 0,C 180,E1 -7104.896,E2 -7104.896} C_VEL
LIN {X 0,Y 474.046,Z 470.368,A -85,B 0,C 180,E1 -7106.599,E2 -7106.599} C_VEL
LIN {X 0,Y 473.795,Z 472.101,A -85,B 0,C 180,E1 -7108.299,E2 -7108.299} C_VEL
LIN {X 0,Y 473.759,Z 472.698,A -85,B 0,C 180,E1 -7109.999,E2 -7109.999} C_VEL
LIN {X 0,Y 473.794,Z 472.149,A -85,B 0,C 180,E1 -7111.699,E2 -7111.699} C_VEL
LIN {X 0,Y 474.044,Z 470.481,A -85,B 0,C 180,E1 -7113.399,E2 -7113.399} C_VEL
LIN {X 0,Y 474.121,Z 467.696,A -85,B 0,C 180,E1 -7115.101,E2 -7115.101} C_VEL
LIN {X 0,Y 474.263,Z 463.584,A -85,B 0,C 180,E1 -7116.85,E2 -7116.85} C_VEL
LIN {X 0,Y 474.523,Z 458.393,A -85,B 0,C 180,E1 -7118.516,E2 -7118.516} C_VEL
LIN {X 0,Y 474.881,Z 451.617,A -85,B 0,C 180,E1 -7120.228,E2 -7120.228} C_VEL
LIN {X 0,Y 475.348,Z 444.351,A -85,B 0,C 180,E1 -7121.728,E2 -7121.728} C_VEL
LIN {X 0,Y 475.94,Z 435.585,A -85,B 0,C 180,E1 -7123.23,E2 -7123.23} C_VEL
LIN {X 0,Y 476.666,Z 424.967,A -85,B 0,C 180,E1 -7124.733,E2 -7124.733} C_VEL
LIN {X 0,Y 477.424,Z 414.053,A -85,B 0,C 180,E1 -7126.021,E2 -7126.021} C_VEL
LIN {X 0,Y 478.185,Z 402.197,A -85,B 0,C 180,E1 -7127.191,E2 -7127.191} C_VEL
LIN {X 0,Y 478.94,Z 388.825,A -85,B 0,C 180,E1 -7128.279,E2 -7128.279} C_VEL
LIN {X 0,Y 479.69,Z 375.875,A -85,B 0,C 180,E1 -7129.135,E2 -7129.135} C_VEL
LIN {X 0,Y 480.27,Z 361.825,A -85,B 0,C 180,E1 -7129.882,E2 -7129.882} C_VEL
LIN {X 0,Y 480.764,Z 347.148,A -85,B 0,C 180,E1 -7130.475,E2 -7130.475} C_VEL
LIN {X 0,Y 481.068,Z 331.739,A -85,B 0,C 180,E1 -7130.915,E2 -7130.915} C_VEL
LIN {X 0,Y 481.352,Z 303.956,A -85,B 0,C 180,E1 -7131.379,E2 -7131.379} C_VEL
LIN {X 0,Y 482.75,Z 179.884,A -85,B 0,C 180,E1 -7133.279,E2 -7133.279} C_VEL
LIN {X 0,Y 481.17,Z 172.246,A -85,B 0,C 180,E1 -7133.485,E2 -7133.485} C_VEL
LIN {X 0,Y 478.749,Z 162.411,A -85,B 0,C 180,E1 -7133.788,E2 -7133.788} C_VEL
LIN {X 0,Y 478.302,Z 158.343,A -85,B 0,C 180,E1 -7134.355,E2 -7134.355} C_VEL
LIN {X 0,Y 474.722,Z 142.979,A -85,B 0,C 180,E1 -7136.841,E2 -7136.841} C_VEL
LIN {X 0,Y 474.602,Z 142.993,A -85,B 0,C 180,E1 -7140.229,E2 -7140.229} C_VEL
LIN {X 0,Y 474.639,Z 142.986,A -85,B 0,C 180,E1 -7143.219,E2 -7143.219} C_VEL
LIN {X 0,Y 474.588,Z 142.99,A -85,B 0,C 180,E1 -7146.322,E2 -7146.322} C_VEL
LIN {X 0,Y 474.612,Z 142.977,A -85,B 0,C 180,E1 -7149.645,E2 -7149.645} C_VEL
LIN {X 0,Y 474.629,Z 142.988,A -85,B 0,C 180,E1 -7152.931,E2 -7152.931} C_VEL
LIN {X 0,Y 474.602,Z 142.99,A -85,B 0,C 180,E1 -7155.894,E2 -7155.894} C_VEL
LIN {X 0,Y 474.633,Z 142.988,A -85,B 0,C 180,E1 -7159.038,E2 -7159.038} C_VEL
LIN {X 0,Y 474.611,Z 142.988,A -85,B 0,C 180,E1 -7161.701,E2 -7161.701} C_VEL
LIN {X 0,Y 474.621,Z 142.987,A -85,B 0,C 180,E1 -7164.725,E2 -7164.725} C_VEL
LIN {X 0,Y 474.628,Z 142.986,A -85,B 0,C 180,E1 -7167.787,E2 -7167.787} C_VEL
LIN {X 0,Y 474.623,Z 142.982,A -85,B 0,C 180,E1 -7170.882,E2 -7170.882} C_VEL
LIN {X 0,Y 474.65,Z 142.981,A -85,B 0,C 180,E1 -7173.628,E2 -7173.628} C_VEL
LIN {X 0,Y 474.625,Z 142.983,A -85,B 0,C 180,E1 -7176.641,E2 -7176.641} C_VEL
LIN {X 0,Y 474.646,Z 142.978,A -85,B 0,C 180,E1 -7180.089,E2 -7180.089} C_VEL
LIN {X 0,Y 474.641,Z 142.984,A -85,B 0,C 180,E1 -7182.774,E2 -7182.774} C_VEL
LIN {X 0,Y 474.638,Z 142.981,A -85,B 0,C 180,E1 -7185.421,E2 -7185.421} C_VEL
LIN {X 0,Y 474.695,Z 142.97,A -85,B 0,C 180,E1 -7188.037,E2 -7188.037} C_VEL
LIN {X 0,Y 474.718,Z 142.972,A -85,B 0,C 180,E1 -7191.486,E2 -7191.486} C_VEL
LIN {X 0,Y 474.769,Z 142.957,A -85,B 0,C 180,E1 -7194.052,E2 -7194.052} C_VEL
LIN {X 0,Y 474.884,Z 142.952,A -85,B 0,C 180,E1 -7197.455,E2 -7197.455} C_VEL
LIN {X 0,Y 474.867,Z 142.951,A -85,B 0,C 180,E1 -7200.848,E2 -7200.848} C_VEL
LIN {X 0,Y 474.884,Z 142.955,A -85,B 0,C 180,E1 -7202.545,E2 -7202.545} C_VEL
LIN {X 0,Y 474.769,Z 142.962,A -85,B 0,C 180,E1 -7205.948,E2 -7205.948} C_VEL
LIN {X 0,Y 474.718,Z 142.973,A -85,B 0,C 180,E1 -7208.514,E2 -7208.514} C_VEL
LIN {X 0,Y 474.694,Z 142.973,A -85,B 0,C 180,E1 -7211.963,E2 -7211.963} C_VEL
LIN {X 0,Y 474.689,Z 142.974,A -85,B 0,C 180,E1 -7215.456,E2 -7215.456} C_VEL
LIN {X 0,Y 474.654,Z 142.974,A -85,B 0,C 180,E1 -7219.011,E2 -7219.011} C_VEL
LIN {X 0,Y 474.587,Z 142.989,A -85,B 0,C 180,E1 -7221.729,E2 -7221.729} C_VEL
LIN {X 0,Y 474.651,Z 142.979,A -85,B 0,C 180,E1 -7224.493,E2 -7224.493} C_VEL
LIN {X 0,Y 474.688,Z 142.977,A -85,B 0,C 180,E1 -7227.339,E2 -7227.339} C_VEL
LIN {X 0,Y 474.595,Z 142.99,A -85,B 0,C 180,E1 -7230.811,E2 -7230.811} C_VEL
LIN {X 0,Y 474.628,Z 142.986,A -85,B 0,C 180,E1 -7233.985,E2 -7233.985} C_VEL
LIN {X 0,Y 474.566,Z 142.993,A -85,B 0,C 180,E1 -7236.901,E2 -7236.901} C_VEL
LIN {X 0,Y 474.618,Z 142.973,A -85,B 0,C 180,E1 -7239.648,E2 -7239.648} C_VEL
LIN {X 0,Y 474.606,Z 142.987,A -85,B 0,C 180,E1 -7242.935,E2 -7242.935} C_VEL
LIN {X 0,Y 474.61,Z 142.993,A -85,B 0,C 180,E1 -7245.897,E2 -7245.897} C_VEL
LIN {X 0,Y 474.639,Z 142.985,A -85,B 0,C 180,E1 -7249.039,E2 -7249.039} C_VEL
LIN {X 0,Y 474.61,Z 142.99,A -85,B 0,C 180,E1 -7251.704,E2 -7251.704} C_VEL
LIN {X 0,Y 474.623,Z 142.982,A -85,B 0,C 180,E1 -7254.727,E2 -7254.727} C_VEL
LIN {X 0,Y 474.698,Z 143.165,A -85,B 0,C 180,E1 -7256.504,E2 -7256.504} C_VEL
LIN {X 0,Y 481.978,Z 167.332,A -85,B 0,C 180,E1 -7259.56,E2 -7259.56} C_VEL
LIN {X 0,Y 482.32,Z 170.378,A -85,B 0,C 180,E1 -7259.898,E2 -7259.898} C_VEL
LIN {X 0,Y 480.246,Z 204.722,A -85,B 0,C 180,E1 -7263.335,E2 -7263.335} C_VEL
LIN {X 0,Y 478.674,Z 236.133,A -85,B 0,C 180,E1 -7266.418,E2 -7266.418} C_VEL
LIN {X 0,Y 478.656,Z 237.884,A -85,B 0,C 180,E1 -7266.553,E2 -7266.553} C_VEL
LIN {X 0,Y 481.429,Z 260.782,A -85,B 0,C 180,E1 -7267.054,E2 -7267.054} C_VEL
LIN {X 0,Y 479.947,Z 404.502,A -85,B 0,C 180,E1 -7269.258,E2 -7269.258} C_VEL
LIN {X 0,Y 479.492,Z 419.909,A -85,B 0,C 180,E1 -7269.65,E2 -7269.65} C_VEL
LIN {X 0,Y 478.916,Z 434.334,A -85,B 0,C 180,E1 -7270.185,E2 -7270.185} C_VEL
LIN {X 0,Y 478.165,Z 449.131,A -85,B 0,C 180,E1 -7270.913,E2 -7270.913} C_VEL
LIN {X 0,Y 477.421,Z 462.851,A -85,B 0,C 180,E1 -7271.772,E2 -7271.772} C_VEL
LIN {X 0,Y 476.625,Z 476.78,A -85,B 0,C 180,E1 -7272.849,E2 -7272.849} C_VEL
LIN {X 0,Y 475.925,Z 489.363,A -85,B 0,C 180,E1 -7274.037,E2 -7274.037} C_VEL
LIN {X 0,Y 475.223,Z 501.687,A -85,B 0,C 180,E1 -7275.44,E2 -7275.44} C_VEL
LIN {X 0,Y 474.717,Z 512.645,A -85,B 0,C 180,E1 -7276.953,E2 -7276.953} C_VEL
LIN {X 0,Y 474.353,Z 521.761,A -85,B 0,C 180,E1 -7278.463,E2 -7278.463} C_VEL
LIN {X 0,Y 474.202,Z 528.316,A -85,B 0,C 180,E1 -7279.757,E2 -7279.757} C_VEL
LIN {X 0,Y 474.024,Z 535.57,A -85,B 0,C 180,E1 -7281.475,E2 -7281.475} C_VEL
LIN {X 0,Y 473.976,Z 541.28,A -85,B 0,C 180,E1 -7283.189,E2 -7283.189} C_VEL
LIN {X 0,Y 473.985,Z 545.591,A -85,B 0,C 180,E1 -7284.897,E2 -7284.897} C_VEL
LIN {X 0,Y 473.99,Z 548.612,A -85,B 0,C 180,E1 -7286.601,E2 -7286.601} C_VEL
LIN {X 0,Y 473.932,Z 550.41,A -85,B 0,C 180,E1 -7288.302,E2 -7288.302} C_VEL
LIN {X 0,Y 474.024,Z 551.033,A -85,B 0,C 180,E1 -7290.001,E2 -7290.001} C_VEL
LIN {X 0,Y 473.932,Z 550.412,A -85,B 0,C 180,E1 -7291.701,E2 -7291.701} C_VEL
LIN {X 0,Y 474.001,Z 548.615,A -85,B 0,C 180,E1 -7293.401,E2 -7293.401} C_VEL
LIN {X 0,Y 473.984,Z 545.588,A -85,B 0,C 180,E1 -7295.105,E2 -7295.105} C_VEL
LIN {X 0,Y 474.018,Z 541.273,A -85,B 0,C 180,E1 -7296.813,E2 -7296.813} C_VEL
LIN {X 0,Y 474.053,Z 535.565,A -85,B 0,C 180,E1 -7298.527,E2 -7298.527} C_VEL
LIN {X 0,Y 474.237,Z 528.314,A -85,B 0,C 180,E1 -7300.245,E2 -7300.245} C_VEL
LIN {X 0,Y 474.385,Z 520.534,A -85,B 0,C 180,E1 -7301.755,E2 -7301.755} C_VEL
LIN {X 0,Y 474.786,Z 511.18,A -85,B 0,C 180,E1 -7303.265,E2 -7303.265} C_VEL
LIN {X 0,Y 475.25,Z 501.668,A -85,B 0,C 180,E1 -7304.561,E2 -7304.561} C_VEL
LIN {X 0,Y 475.832,Z 490.369,A -85,B 0,C 180,E1 -7305.858,E2 -7305.858} C_VEL
LIN {X 0,Y 476.536,Z 477.993,A -85,B 0,C 180,E1 -7307.046,E2 -7307.046} C_VEL
LIN {X 0,Y 477.334,Z 464.382,A -85,B 0,C 180,E1 -7308.122,E2 -7308.122} C_VEL
LIN {X 0,Y 478.079,Z 451,A -85,B 0,C 180,E1 -7308.982,E2 -7308.982} C_VEL
LIN {X 0,Y 478.823,Z 436.28,A -85,B 0,C 180,E1 -7309.731,E2 -7309.731} C_VEL
LIN {X 0,Y 479.455,Z 420.828,A -85,B 0,C 180,E1 -7310.32,E2 -7310.32} C_VEL
LIN {X 0,Y 479.984,Z 405.738,A -85,B 0,C 180,E1 -7310.715,E2 -7310.715} C_VEL
LIN {X 0,Y 481.402,Z 266.68,A -85,B 0,C 180,E1 -7312.852,E2 -7312.852} C_VEL
LIN {X 0,Y 481.24,Z 257.779,A -85,B 0,C 180,E1 -7313,E2 -7313} C_VEL
LIN {X 0,Y 478.572,Z 237.153,A -85,B 0,C 180,E1 -7313.475,E2 -7313.475} C_VEL
LIN {X 0,Y 480.022,Z 212.726,A -85,B 0,C 180,E1 -7315.939,E2 -7315.939} C_VEL
LIN {X 0,Y 482.279,Z 182.624,A -85,B 0,C 180,E1 -7319.126,E2 -7319.126} C_VEL
LIN {X 0,Y 483.416,Z 170.36,A -85,B 0,C 180,E1 -7320.486,E2 -7320.486} C_VEL
LIN {X 0,Y 480.622,Z 160.279,A -85,B 0,C 180,E1 -7321.993,E2 -7321.993} C_VEL
LIN {X 0,Y 477.26,Z 150.251,A -85,B 0,C 180,E1 -7323.696,E2 -7323.696} C_VEL
LIN {X 0,Y 474.634,Z 142.992,A -85,B 0,C 180,E1 -7325.112,E2 -7325.112} C_VEL
LIN {X 0,Y 474.61,Z 142.992,A -85,B 0,C 180,E1 -7328.458,E2 -7328.458} C_VEL
LIN {X 0,Y 474.593,Z 142.995,A -85,B 0,C 180,E1 -7331.789,E2 -7331.789} C_VEL
LIN {X 0,Y 474.615,Z 142.993,A -85,B 0,C 180,E1 -7335.299,E2 -7335.299} C_VEL
LIN {X 0,Y 474.583,Z 142.994,A -85,B 0,C 180,E1 -7338.211,E2 -7338.211} C_VEL
LIN {X 0,Y 474.586,Z 142.996,A -85,B 0,C 180,E1 -7341.54,E2 -7341.54} C_VEL
LIN {X 0,Y 474.612,Z 142.993,A -85,B 0,C 180,E1 -7344.725,E2 -7344.725} C_VEL
LIN {X 0,Y 474.62,Z 142.992,A -85,B 0,C 180,E1 -7347.787,E2 -7347.787} C_VEL
LIN {X 0,Y 474.632,Z 143.111,A -85,B 0,C 180,E1 -7350.414,E2 -7350.414} C_VEL
LIN {X 0,Y 477.914,Z 153.945,A -85,B 0,C 180,E1 -7353.116,E2 -7353.116} C_VEL
LIN {X 0,Y 480.371,Z 164.294,A -85,B 0,C 180,E1 -7355.438,E2 -7355.438} C_VEL
LIN {X 0,Y 480.559,Z 167.413,A -85,B 0,C 180,E1 -7356.057,E2 -7356.057} C_VEL
LIN {X 0,Y 479.264,Z 184.577,A -85,B 0,C 180,E1 -7359.17,E2 -7359.17} C_VEL
LIN {X 0,Y 478.139,Z 202.847,A -85,B 0,C 180,E1 -7362.37,E2 -7362.37} C_VEL
LIN {X 0,Y 480.673,Z 213.65,A -85,B 0,C 180,E1 -7362.771,E2 -7362.771} C_VEL
LIN {X 0,Y 478.374,Z 303.891,A -85,B 0,C 180,E1 -7364.666,E2 -7364.666} C_VEL
LIN {X 0,Y 478.127,Z 321.013,A -85,B 0,C 180,E1 -7365.067,E2 -7365.067} C_VEL
LIN {X 0,Y 477.89,Z 334.578,A -85,B 0,C 180,E1 -7365.577,E2 -7365.577} C_VEL
LIN {X 0,Y 477.62,Z 346.87,A -85,B 0,C 180,E1 -7366.21,E2 -7366.21} C_VEL
LIN {X 0,Y 477.168,Z 358.683,A -85,B 0,C 180,E1 -7366.992,E2 -7366.992} C_VEL
LIN {X 0,Y 476.733,Z 370.398,A -85,B 0,C 180,E1 -7367.981,E2 -7367.981} C_VEL
LIN {X 0,Y 476.37,Z 379.627,A -85,B 0,C 180,E1 -7368.943,E2 -7368.943} C_VEL
LIN {X 0,Y 476.025,Z 388.087,A -85,B 0,C 180,E1 -7370.01,E2 -7370.01} C_VEL
LIN {X 0,Y 475.557,Z 396.314,A -85,B 0,C 180,E1 -7371.287,E2 -7371.287} C_VEL
LIN {X 0,Y 475.223,Z 403.071,A -85,B 0,C 180,E1 -7372.599,E2 -7372.599} C_VEL
LIN {X 0,Y 474.945,Z 408.947,A -85,B 0,C 180,E1 -7374.055,E2 -7374.055} C_VEL
LIN {X 0,Y 474.785,Z 412.818,A -85,B 0,C 180,E1 -7375.33,E2 -7375.33} C_VEL
LIN {X 0,Y 474.642,Z 415.631,A -85,B 0,C 180,E1 -7376.605,E2 -7376.605} C_VEL
LIN {X 0,Y 474.561,Z 416.965,A -85,B 0,C 180,E1 -7377.454,E2 -7377.454} C_VEL
LIN {X 0,Y 474.565,Z 417.854,A -85,B 0,C 180,E1 -7378.303,E2 -7378.303} C_VEL
LIN {X 0,Y 474.491,Z 418.363,A -85,B 0,C 180,E1 -7379.151,E2 -7379.151} C_VEL
LIN {X 0,Y 474.46,Z 418.474,A -85,B 0,C 180,E1 -7380,E2 -7380} C_VEL
LIN {X 0,Y 474.475,Z 418.147,A -85,B 0,C 180,E1 -7380.849,E2 -7380.849} C_VEL
LIN {X 0,Y 474.397,Z 417.422,A -85,B 0,C 180,E1 -7381.698,E2 -7381.698} C_VEL
LIN {X 0,Y 474.507,Z 416.276,A -85,B 0,C 180,E1 -7382.547,E2 -7382.547} C_VEL
LIN {X 0,Y 474.446,Z 413.792,A -85,B 0,C 180,E1 -7383.822,E2 -7383.822} C_VEL
LIN {X 0,Y 474.569,Z 410.288,A -85,B 0,C 180,E1 -7385.098,E2 -7385.098} C_VEL
LIN {X 0,Y 474.818,Z 405.687,A -85,B 0,C 180,E1 -7386.374,E2 -7386.374} C_VEL
LIN {X 0,Y 474.97,Z 399.883,A -85,B 0,C 180,E1 -7387.653,E2 -7387.653} C_VEL
LIN {X 0,Y 475.293,Z 392.65,A -85,B 0,C 180,E1 -7388.932,E2 -7388.932} C_VEL
LIN {X 0,Y 475.596,Z 383.626,A -85,B 0,C 180,E1 -7390.214,E2 -7390.214} C_VEL
LIN {X 0,Y 475.935,Z 373.392,A -85,B 0,C 180,E1 -7391.391,E2 -7391.391} C_VEL
LIN {X 0,Y 476.395,Z 363.006,A -85,B 0,C 180,E1 -7392.352,E2 -7392.352} C_VEL
LIN {X 0,Y 476.727,Z 350.875,A -85,B 0,C 180,E1 -7393.255,E2 -7393.255} C_VEL
LIN {X 0,Y 477.027,Z 338.777,A -85,B 0,C 180,E1 -7393.961,E2 -7393.961} C_VEL
LIN {X 0,Y 477.272,Z 325.8,A -85,B 0,C 180,E1 -7394.524,E2 -7394.524} C_VEL
LIN {X 0,Y 477.489,Z 312.475,A -85,B 0,C 180,E1 -7394.926,E2 -7394.926} C_VEL
LIN {X 0,Y 478.603,Z 210.742,A -85,B 0,C 180,E1 -7396.724,E2 -7396.724} C_VEL
LIN {X 0,Y 476.309,Z 198.501,A -85,B 0,C 180,E1 -7397.045,E2 -7397.045} C_VEL
LIN {X 0,Y 477.022,Z 179.081,A -85,B 0,C 180,E1 -7400.257,E2 -7400.257} C_VEL
LIN {X 0,Y 477.782,Z 160.311,A -85,B 0,C 180,E1 -7403.401,E2 -7403.401} C_VEL
LIN {X 0,Y 477.683,Z 156.999,A -85,B 0,C 180,E1 -7403.977,E2 -7403.977} C_VEL
LIN {X 0,Y 474.665,Z 142.985,A -85,B 0,C 180,E1 -7406.579,E2 -7406.579} C_VEL
LIN {X 0,Y 474.612,Z 142.993,A -85,B 0,C 180,E1 -7409.253,E2 -7409.253} C_VEL
LIN {X 0,Y 474.62,Z 142.987,A -85,B 0,C 180,E1 -7412.43,E2 -7412.43} C_VEL
LIN {X 0,Y 474.616,Z 142.992,A -85,B 0,C 180,E1 -7415.468,E2 -7415.468} C_VEL
LIN {X 0,Y 474.614,Z 142.987,A -85,B 0,C 180,E1 -7418.457,E2 -7418.457} C_VEL
LIN {X 0,Y 474.619,Z 142.988,A -85,B 0,C 180,E1 -7421.786,E2 -7421.786} C_VEL
LIN {X 0,Y 474.621,Z 142.991,A -85,B 0,C 180,E1 -7425.297,E2 -7425.297} C_VEL
LIN {X 0,Y 474.625,Z 142.986,A -85,B 0,C 180,E1 -7428.214,E2 -7428.214} C_VEL
LIN {X 0,Y 474.615,Z 142.99,A -85,B 0,C 180,E1 -7431.542,E2 -7431.542} C_VEL
LIN {X 0,Y 474.587,Z 142.994,A -85,B 0,C 180,E1 -7433.587,E2 -7433.587} C_VEL
LIN {X 0,Y 473.964,Z 143.074,A -85,B 0,C 180,E1 -7434.295,E2 -7434.295} C_VEL
LIN {X 0,Y 471.149,Z 143.426,A -85,B 0,C 180,E1 -7435.447,E2 -7435.447} C_VEL
LIN {X 0,Y 468.734,Z 143.728,A -85,B 0,C 180,E1 -7436.375,E2 -7436.375} C_VEL
LIN {X 0,Y 467.678,Z 143.857,A -85,B 0,C 180,E1 -7437.092,E2 -7437.092} C_VEL
LIN {X 0,Y 467.583,Z 143.867,A -85,B 0,C 180,E1 -7437.335,E2 -7437.335} C_VEL
LIN {X 0,Y 467.573,Z 143.87,A -85,B 0,C 180,E1 -7440.667,E2 -7440.667} C_VEL
LIN {X 0,Y 467.709,Z 144.017,A -85,B 0,C 180,E1 -7442.952,E2 -7442.952} C_VEL
LIN {X 0,Y 471.378,Z 159.331,A -85,B 0,C 180,E1 -7445.434,E2 -7445.434} C_VEL
LIN {X 0,Y 472.071,Z 163.195,A -85,B 0,C 180,E1 -7445.969,E2 -7445.969} C_VEL
LIN {X 0,Y 476.155,Z 179.85,A -85,B 0,C 180,E1 -7446.464,E2 -7446.464} C_VEL
LIN {X 0,Y 474.962,Z 293.115,A -85,B 0,C 180,E1 -7448.231,E2 -7448.231} C_VEL
LIN {X 0,Y 474.49,Z 330.793,A -85,B 0,C 180,E1 -7448.844,E2 -7448.844} C_VEL
LIN {X 0,Y 474.165,Z 346.171,A -85,B 0,C 180,E1 -7449.27,E2 -7449.27} C_VEL
LIN {X 0,Y 473.707,Z 360.235,A -85,B 0,C 180,E1 -7449.826,E2 -7449.826} C_VEL
LIN {X 0,Y 473.072,Z 374.839,A -85,B 0,C 180,E1 -7450.584,E2 -7450.584} C_VEL
LIN {X 0,Y 472.357,Z 388.102,A -85,B 0,C 180,E1 -7451.455,E2 -7451.455} C_VEL
LIN {X 0,Y 471.537,Z 400.578,A -85,B 0,C 180,E1 -7452.455,E2 -7452.455} C_VEL
LIN {X 0,Y 470.757,Z 412.71,A -85,B 0,C 180,E1 -7453.632,E2 -7453.632} C_VEL
LIN {X 0,Y 469.996,Z 423.087,A -85,B 0,C 180,E1 -7454.829,E2 -7454.829} C_VEL
LIN {X 0,Y 469.272,Z 432.681,A -85,B 0,C 180,E1 -7456.135,E2 -7456.135} C_VEL
LIN {X 0,Y 468.667,Z 441.476,A -85,B 0,C 180,E1 -7457.555,E2 -7457.555} C_VEL
LIN {X 0,Y 468.079,Z 449.842,A -85,B 0,C 180,E1 -7459.181,E2 -7459.181} C_VEL
LIN {X 0,Y 467.622,Z 457.088,A -85,B 0,C 180,E1 -7460.919,E2 -7460.919} C_VEL
LIN {X 0,Y 467.304,Z 462.831,A -85,B 0,C 180,E1 -7462.654,E2 -7462.654} C_VEL
LIN {X 0,Y 467.072,Z 466.223,A -85,B 0,C 180,E1 -7463.953,E2 -7463.953} C_VEL
LIN {X 0,Y 467.008,Z 469.672,A -85,B 0,C 180,E1 -7465.684,E2 -7465.684} C_VEL
LIN {X 0,Y 466.845,Z 471.959,A -85,B 0,C 180,E1 -7467.41,E2 -7467.41} C_VEL
LIN {X 0,Y 466.691,Z 473.13,A -85,B 0,C 180,E1 -7469.136,E2 -7469.136} C_VEL
LIN {X 0,Y 466.691,Z 473.146,A -85,B 0,C 180,E1 -7470.862,E2 -7470.862} C_VEL
LIN {X 0,Y 466.845,Z 472.038,A -85,B 0,C 180,E1 -7472.587,E2 -7472.587} C_VEL
LIN {X 0,Y 466.999,Z 469.819,A -85,B 0,C 180,E1 -7474.314,E2 -7474.314} C_VEL
LIN {X 0,Y 467.065,Z 466.446,A -85,B 0,C 180,E1 -7476.045,E2 -7476.045} C_VEL
LIN {X 0,Y 467.36,Z 461.804,A -85,B 0,C 180,E1 -7477.777,E2 -7477.777} C_VEL
LIN {X 0,Y 467.699,Z 455.78,A -85,B 0,C 180,E1 -7479.513,E2 -7479.513} C_VEL
LIN {X 0,Y 468.18,Z 448.196,A -85,B 0,C 180,E1 -7481.252,E2 -7481.252} C_VEL
LIN {X 0,Y 468.715,Z 440.264,A -85,B 0,C 180,E1 -7482.749,E2 -7482.749} C_VEL
LIN {X 0,Y 469.358,Z 431.857,A -85,B 0,C 180,E1 -7484.081,E2 -7484.081} C_VEL
LIN {X 0,Y 470.191,Z 420.33,A -85,B 0,C 180,E1 -7485.606,E2 -7485.606} C_VEL
LIN {X 0,Y 470.989,Z 409.126,A -85,B 0,C 180,E1 -7486.838,E2 -7486.838} C_VEL
LIN {X 0,Y 471.814,Z 396.624,A -85,B 0,C 180,E1 -7487.98,E2 -7487.98} C_VEL
LIN {X 0,Y 472.655,Z 383.247,A -85,B 0,C 180,E1 -7488.98,E2 -7488.98} C_VEL
LIN {X 0,Y 473.326,Z 368.706,A -85,B 0,C 180,E1 -7489.854,E2 -7489.854} C_VEL
LIN {X 0,Y 473.915,Z 354.031,A -85,B 0,C 180,E1 -7490.535,E2 -7490.535} C_VEL
LIN {X 0,Y 474.35,Z 339.655,A -85,B 0,C 180,E1 -7491.027,E2 -7491.027} C_VEL
LIN {X 0,Y 474.594,Z 325.466,A -85,B 0,C 180,E1 -7491.356,E2 -7491.356} C_VEL
LIN {X 0,Y 476.25,Z 180.419,A -85,B 0,C 180,E1 -7493.615,E2 -7493.615} C_VEL
LIN {X 0,Y 472.024,Z 162.884,A -85,B 0,C 180,E1 -7494.149,E2 -7494.149} C_VEL
LIN {X 0,Y 469.788,Z 152.634,A -85,B 0,C 180,E1 -7495.71,E2 -7495.71} C_VEL
LIN {X 0,Y 467.673,Z 143.859,A -85,B 0,C 180,E1 -7497.188,E2 -7497.188} C_VEL
LIN {X 0,Y 467.566,Z 143.87,A -85,B 0,C 180,E1 -7500.732,E2 -7500.732} C_VEL
LIN {X 0,Y 467.583,Z 143.868,A -85,B 0,C 180,E1 -7503.787,E2 -7503.787} C_VEL
LIN {X 0,Y 467.545,Z 143.871,A -85,B 0,C 180,E1 -7507.186,E2 -7507.186} C_VEL
LIN {X 0,Y 467.57,Z 143.852,A -85,B 0,C 180,E1 -7510.264,E2 -7510.264} C_VEL
LIN {X 0,Y 467.58,Z 143.864,A -85,B 0,C 180,E1 -7512.566,E2 -7512.566} C_VEL
LIN {X 0,Y 467.563,Z 143.866,A -85,B 0,C 180,E1 -7515.052,E2 -7515.052} C_VEL
LIN {X 0,Y 467.581,Z 143.864,A -85,B 0,C 180,E1 -7517.439,E2 -7517.439} C_VEL
LIN {X 0,Y 467.611,Z 143.861,A -85,B 0,C 180,E1 -7520.858,E2 -7520.858} C_VEL
LIN {X 0,Y 467.554,Z 143.865,A -85,B 0,C 180,E1 -7524.259,E2 -7524.259} C_VEL
LIN {X 0,Y 467.573,Z 143.869,A -85,B 0,C 180,E1 -7527.32,E2 -7527.32} C_VEL
LIN {X 0,Y 467.569,Z 143.858,A -85,B 0,C 180,E1 -7530.665,E2 -7530.665} C_VEL
LIN {X 0,Y 467.607,Z 143.863,A -85,B 0,C 180,E1 -7533.199,E2 -7533.199} C_VEL
LIN {X 0,Y 467.582,Z 143.859,A -85,B 0,C 180,E1 -7536.467,E2 -7536.467} C_VEL
LIN {X 0,Y 467.613,Z 143.854,A -85,B 0,C 180,E1 -7539.777,E2 -7539.777} C_VEL
LIN {X 0,Y 467.599,Z 143.858,A -85,B 0,C 180,E1 -7542.506,E2 -7542.506} C_VEL
LIN {X 0,Y 467.596,Z 143.86,A -85,B 0,C 180,E1 -7545.196,E2 -7545.196} C_VEL
LIN {X 0,Y 467.646,Z 143.847,A -85,B 0,C 180,E1 -7547.854,E2 -7547.854} C_VEL
LIN {X 0,Y 467.671,Z 143.85,A -85,B 0,C 180,E1 -7551.357,E2 -7551.357} C_VEL
LIN {X 0,Y 467.733,Z 143.833,A -85,B 0,C 180,E1 -7553.962,E2 -7553.962} C_VEL
LIN {X 0,Y 467.85,Z 143.829,A -85,B 0,C 180,E1 -7557.417,E2 -7557.417} C_VEL
LIN {X 0,Y 467.871,Z 143.817,A -85,B 0,C 180,E1 -7560,E2 -7560} C_VEL
LIN {X 0,Y 467.849,Z 143.832,A -85,B 0,C 180,E1 -7562.583,E2 -7562.583} C_VEL
LIN {X 0,Y 467.733,Z 143.839,A -85,B 0,C 180,E1 -7566.037,E2 -7566.037} C_VEL
LIN {X 0,Y 467.671,Z 143.852,A -85,B 0,C 180,E1 -7568.643,E2 -7568.643} C_VEL
LIN {X 0,Y 467.645,Z 143.852,A -85,B 0,C 180,E1 -7572.146,E2 -7572.146} C_VEL
LIN {X 0,Y 467.644,Z 143.852,A -85,B 0,C 180,E1 -7575.695,E2 -7575.695} C_VEL
LIN {X 0,Y 467.606,Z 143.853,A -85,B 0,C 180,E1 -7578.765,E2 -7578.765} C_VEL
LIN {X 0,Y 467.573,Z 143.862,A -85,B 0,C 180,E1 -7581.27,E2 -7581.27} C_VEL
LIN {X 0,Y 467.565,Z 143.863,A -85,B 0,C 180,E1 -7583.944,E2 -7583.944} C_VEL
LIN {X 0,Y 467.606,Z 143.862,A -85,B 0,C 180,E1 -7586.801,E2 -7586.801} C_VEL
LIN {X 0,Y 467.544,Z 143.862,A -85,B 0,C 180,E1 -7589.739,E2 -7589.739} C_VEL
LIN {X 0,Y 467.574,Z 143.864,A -85,B 0,C 180,E1 -7592.759,E2 -7592.759} C_VEL
LIN {X 0,Y 467.547,Z 143.869,A -85,B 0,C 180,E1 -7595.89,E2 -7595.89} C_VEL
LIN {X 0,Y 467.573,Z 143.851,A -85,B 0,C 180,E1 -7599.146,E2 -7599.146} C_VEL
LIN {X 0,Y 467.578,Z 143.865,A -85,B 0,C 180,E1 -7602.568,E2 -7602.568} C_VEL
LIN {X 0,Y 467.562,Z 143.866,A -85,B 0,C 180,E1 -7605.054,E2 -7605.054} C_VEL
LIN {X 0,Y 467.617,Z 143.86,A -85,B 0,C 180,E1 -7607.445,E2 -7607.445} C_VEL
LIN {X 0,Y 467.593,Z 143.86,A -85,B 0,C 180,E1 -7610.858,E2 -7610.858} C_VEL
LIN {X 0,Y 467.556,Z 143.866,A -85,B 0,C 180,E1 -7614.262,E2 -7614.262} C_VEL
LIN {X 0,Y 467.624,Z 144.045,A -85,B 0,C 180,E1 -7616.132,E2 -7616.132} C_VEL
LIN {X 0,Y 474.751,Z 167.541,A -85,B 0,C 180,E1 -7619.16,E2 -7619.16} C_VEL
LIN {X 0,Y 475.602,Z 170.613,A -85,B 0,C 180,E1 -7619.539,E2 -7619.539} C_VEL
LIN {X 0,Y 474.321,Z 191.722,A -85,B 0,C 180,E1 -7621.698,E2 -7621.698} C_VEL
LIN {X 0,Y 472.296,Z 228.364,A -85,B 0,C 180,E1 -7625.378,E2 -7625.378} C_VEL
LIN {X 0,Y 471.831,Z 236.387,A -85,B 0,C 180,E1 -7626.171,E2 -7626.171} C_VEL
LIN {X 0,Y 474.864,Z 261.33,A -85,B 0,C 180,E1 -7626.734,E2 -7626.734} C_VEL
LIN {X 0,Y 473.4,Z 399.576,A -85,B 0,C 180,E1 -7628.872,E2 -7628.872} C_VEL
LIN {X 0,Y 472.996,Z 415.193,A -85,B 0,C 180,E1 -7629.227,E2 -7629.227} C_VEL
LIN {X 0,Y 472.386,Z 429.059,A -85,B 0,C 180,E1 -7629.693,E2 -7629.693} C_VEL
LIN {X 0,Y 471.712,Z 443.596,A -85,B 0,C 180,E1 -7630.358,E2 -7630.358} C_VEL
LIN {X 0,Y 470.871,Z 457.503,A -85,B 0,C 180,E1 -7631.171,E2 -7631.171} C_VEL
LIN {X 0,Y 470.109,Z 470.994,A -85,B 0,C 180,E1 -7632.155,E2 -7632.155} C_VEL
LIN {X 0,Y 469.386,Z 483.378,A -85,B 0,C 180,E1 -7633.25,E2 -7633.25} C_VEL
LIN {X 0,Y 468.597,Z 495.705,A -85,B 0,C 180,E1 -7634.562,E2 -7634.562} C_VEL
LIN {X 0,Y 467.998,Z 506.06,A -85,B 0,C 180,E1 -7635.877,E2 -7635.877} C_VEL
LIN {X 0,Y 467.516,Z 516.186,A -85,B 0,C 180,E1 -7637.412,E2 -7637.412} C_VEL
LIN {X 0,Y 467.211,Z 524.591,A -85,B 0,C 180,E1 -7638.944,E2 -7638.944} C_VEL
LIN {X 0,Y 466.949,Z 531.553,A -85,B 0,C 180,E1 -7640.471,E2 -7640.471} C_VEL
LIN {X 0,Y 466.901,Z 538.02,A -85,B 0,C 180,E1 -7642.215,E2 -7642.215} C_VEL
LIN {X 0,Y 466.9,Z 543.016,A -85,B 0,C 180,E1 -7643.953,E2 -7643.953} C_VEL
LIN {X 0,Y 466.963,Z 546.675,A -85,B 0,C 180,E1 -7645.685,E2 -7645.685} C_VEL
LIN {X 0,Y 466.92,Z 549.078,A -85,B 0,C 180,E1 -7647.413,E2 -7647.413} C_VEL
LIN {X 0,Y 466.945,Z 550.29,A -85,B 0,C 180,E1 -7649.139,E2 -7649.139} C_VEL
LIN {X 0,Y 466.918,Z 550.289,A -85,B 0,C 180,E1 -7650.864,E2 -7650.864} C_VEL
LIN {X 0,Y 466.922,Z 549.08,A -85,B 0,C 180,E1 -7652.589,E2 -7652.589} C_VEL
LIN {X 0,Y 466.942,Z 546.674,A -85,B 0,C 180,E1 -7654.317,E2 -7654.317} C_VEL
LIN {X 0,Y 466.898,Z 543.008,A -85,B 0,C 180,E1 -7656.049,E2 -7656.049} C_VEL
LIN {X 0,Y 466.927,Z 538.01,A -85,B 0,C 180,E1 -7657.787,E2 -7657.787} C_VEL
LIN {X 0,Y 466.997,Z 531.55,A -85,B 0,C 180,E1 -7659.53,E2 -7659.53} C_VEL
LIN {X 0,Y 467.221,Z 524.584,A -85,B 0,C 180,E1 -7661.058,E2 -7661.058} C_VEL
LIN {X 0,Y 467.548,Z 516.431,A -85,B 0,C 180,E1 -7662.546,E2 -7662.546} C_VEL
LIN {X 0,Y 468.019,Z 506.039,A -85,B 0,C 180,E1 -7664.125,E2 -7664.125} C_VEL
LIN {X 0,Y 468.63,Z 495.68,A -85,B 0,C 180,E1 -7665.439,E2 -7665.439} C_VEL
LIN {X 0,Y 469.359,Z 483.553,A -85,B 0,C 180,E1 -7666.731,E2 -7666.731} C_VEL
LIN {X 0,Y 470.094,Z 470.944,A -85,B 0,C 180,E1 -7667.848,E2 -7667.848} C_VEL
LIN {X 0,Y 470.915,Z 457.46,A -85,B 0,C 180,E1 -7668.829,E2 -7668.829} C_VEL
LIN {X 0,Y 471.766,Z 443.529,A -85,B 0,C 180,E1 -7669.642,E2 -7669.642} C_VEL
LIN {X 0,Y 472.445,Z 429.02,A -85,B 0,C 180,E1 -7670.303,E2 -7670.303} C_VEL
LIN {X 0,Y 473.023,Z 413.915,A -85,B 0,C 180,E1 -7670.809,E2 -7670.809} C_VEL
LIN {X 0,Y 473.421,Z 399.344,A -85,B 0,C 180,E1 -7671.129,E2 -7671.129} C_VEL
LIN {X 0,Y 474.892,Z 261.012,A -85,B 0,C 180,E1 -7673.267,E2 -7673.267} C_VEL
LIN {X 0,Y 472.449,Z 240.839,A -85,B 0,C 180,E1 -7673.717,E2 -7673.717} C_VEL
LIN {X 0,Y 471.884,Z 236.91,A -85,B 0,C 180,E1 -7673.829,E2 -7673.829} C_VEL
LIN {X 0,Y 473.447,Z 212.741,A -85,B 0,C 180,E1 -7676.327,E2 -7676.327} C_VEL
LIN {X 0,Y 475.914,Z 183.513,A -85,B 0,C 180,E1 -7679.505,E2 -7679.505} C_VEL
LIN {X 0,Y 476.921,Z 172.285,A -85,B 0,C 180,E1 -7680.798,E2 -7680.798} C_VEL
LIN {X 0,Y 474.129,Z 162.424,A -85,B 0,C 180,E1 -7682.338,E2 -7682.338} C_VEL
LIN {X 0,Y 470.916,Z 152.804,A -85,B 0,C 180,E1 -7684.044,E2 -7684.044} C_VEL
LIN {X 0,Y 467.542,Z 143.874,A -85,B 0,C 180,E1 -7685.925,E2 -7685.925} C_VEL
LIN {X 0,Y 467.554,Z 143.871,A -85,B 0,C 180,E1 -7689.148,E2 -7689.148} C_VEL
LIN {X 0,Y 467.561,Z 143.872,A -85,B 0,C 180,E1 -7691.406,E2 -7691.406} C_VEL
LIN {X 0,Y 467.564,Z 143.871,A -85,B 0,C 180,E1 -7695.052,E2 -7695.052} C_VEL
LIN {X 0,Y 467.552,Z 143.87,A -85,B 0,C 180,E1 -7698.728,E2 -7698.728} C_VEL
LIN {X 0,Y 467.539,Z 143.873,A -85,B 0,C 180,E1 -7701.953,E2 -7701.953} C_VEL
LIN {X 0,Y 467.553,Z 143.872,A -85,B 0,C 180,E1 -7705.166,E2 -7705.166} C_VEL
LIN {X 0,Y 467.552,Z 143.873,A -85,B 0,C 180,E1 -7708.258,E2 -7708.258} C_VEL
LIN {X 0,Y 467.539,Z 143.886,A -85,B 0,C 180,E1 -7709.577,E2 -7709.577} C_VEL
LIN {X 0,Y 470.601,Z 153.612,A -85,B 0,C 180,E1 -7712.175,E2 -7712.175} C_VEL
LIN {X 0,Y 473.11,Z 163.274,A -85,B 0,C 180,E1 -7714.482,E2 -7714.482} C_VEL
LIN {X 0,Y 474.064,Z 168.912,A -85,B 0,C 180,E1 -7715.708,E2 -7715.708} C_VEL
LIN {X 0,Y 472.969,Z 182.265,A -85,B 0,C 180,E1 -7718.193,E2 -7718.193} C_VEL
LIN {X 0,Y 471.588,Z 200.825,A -85,B 0,C 180,E1 -7721.538,E2 -7721.538} C_VEL
LIN {X 0,Y 471.444,Z 203.24,A -85,B 0,C 180,E1 -7721.965,E2 -7721.965} C_VEL
LIN {X 0,Y 474.248,Z 215.005,A -85,B 0,C 180,E1 -7722.432,E2 -7722.432} C_VEL
LIN {X 0,Y 471.672,Z 306.061,A -85,B 0,C 180,E1 -7724.415,E2 -7724.415} C_VEL
LIN {X 0,Y 471.407,Z 322.568,A -85,B 0,C 180,E1 -7724.821,E2 -7724.821} C_VEL
LIN {X 0,Y 471.181,Z 335.25,A -85,B 0,C 180,E1 -7725.311,E2 -7725.311} C_VEL
LIN {X 0,Y 470.898,Z 347.596,A -85,B 0,C 180,E1 -7725.957,E2 -7725.957} C_VEL
LIN {X 0,Y 470.427,Z 358.827,A -85,B 0,C 180,E1 -7726.702,E2 -7726.702} C_VEL
LIN {X 0,Y 470.041,Z 369.457,A -85,B 0,C 180,E1 -7727.588,E2 -7727.588} C_VEL
LIN {X 0,Y 469.602,Z 379.005,A -85,B 0,C 180,E1 -7728.563,E2 -7728.563} C_VEL
LIN {X 0,Y 469.207,Z 387.732,A -85,B 0,C 180,E1 -7729.645,E2 -7729.645} C_VEL
LIN {X 0,Y 468.745,Z 396.285,A -85,B 0,C 180,E1 -7730.942,E2 -7730.942} C_VEL
LIN {X 0,Y 468.321,Z 403.11,A -85,B 0,C 180,E1 -7732.238,E2 -7732.238} C_VEL
LIN {X 0,Y 468.084,Z 408.526,A -85,B 0,C 180,E1 -7733.534,E2 -7733.534} C_VEL
LIN {X 0,Y 467.817,Z 412.757,A -85,B 0,C 180,E1 -7734.829,E2 -7734.829} C_VEL
LIN {X 0,Y 467.677,Z 414.962,A -85,B 0,C 180,E1 -7735.691,E2 -7735.691} C_VEL
LIN {X 0,Y 467.645,Z 416.725,A -85,B 0,C 180,E1 -7736.554,E2 -7736.554} C_VEL
LIN {X 0,Y 467.572,Z 418.037,A -85,B 0,C 180,E1 -7737.416,E2 -7737.416} C_VEL
LIN {X 0,Y 467.55,Z 418.914,A -85,B 0,C 180,E1 -7738.277,E2 -7738.277} C_VEL
LIN {X 0,Y 467.472,Z 419.404,A -85,B 0,C 180,E1 -7739.139,E2 -7739.139} C_VEL
LIN {X 0,Y 467.439,Z 419.493,A -85,B 0,C 180,E1 -7740,E2 -7740} C_VEL
LIN {X 0,Y 467.454,Z 419.138,A -85,B 0,C 180,E1 -7740.862,E2 -7740.862} C_VEL
LIN {X 0,Y 467.374,Z 418.389,A -85,B 0,C 180,E1 -7741.723,E2 -7741.723} C_VEL
LIN {X 0,Y 467.487,Z 417.221,A -85,B 0,C 180,E1 -7742.585,E2 -7742.585} C_VEL
LIN {X 0,Y 467.425,Z 414.691,A -85,B 0,C 180,E1 -7743.88,E2 -7743.88} C_VEL
LIN {X 0,Y 467.56,Z 411.137,A -85,B 0,C 180,E1 -7745.174,E2 -7745.174} C_VEL
LIN {X 0,Y 467.815,Z 406.483,A -85,B 0,C 180,E1 -7746.47,E2 -7746.47} C_VEL
LIN {X 0,Y 467.996,Z 400.621,A -85,B 0,C 180,E1 -7747.768,E2 -7747.768} C_VEL
LIN {X 0,Y 468.318,Z 393.321,A -85,B 0,C 180,E1 -7749.066,E2 -7749.066} C_VEL
LIN {X 0,Y 468.64,Z 384.211,A -85,B 0,C 180,E1 -7750.367,E2 -7750.367} C_VEL
LIN {X 0,Y 468.996,Z 373.897,A -85,B 0,C 180,E1 -7751.562,E2 -7751.562} C_VEL
LIN {X 0,Y 469.478,Z 363.399,A -85,B 0,C 180,E1 -7752.537,E2 -7752.537} C_VEL
LIN {X 0,Y 469.805,Z 351.576,A -85,B 0,C 180,E1 -7753.425,E2 -7753.425} C_VEL
LIN {X 0,Y 470.135,Z 338.914,A -85,B 0,C 180,E1 -7754.169,E2 -7754.169} C_VEL
LIN {X 0,Y 470.403,Z 325.737,A -85,B 0,C 180,E1 -7754.741,E2 -7754.741} C_VEL
LIN {X 0,Y 470.624,Z 312.149,A -85,B 0,C 180,E1 -7755.149,E2 -7755.149} C_VEL
LIN {X 0,Y 471.856,Z 212.009,A -85,B 0,C 180,E1 -7756.952,E2 -7756.952} C_VEL
LIN {X 0,Y 469.392,Z 198.628,A -85,B 0,C 180,E1 -7757.325,E2 -7757.325} C_VEL
LIN {X 0,Y 470.259,Z 177.889,A -85,B 0,C 180,E1 -7760.79,E2 -7760.79} C_VEL
LIN {X 0,Y 470.96,Z 160.375,A -85,B 0,C 180,E1 -7763.761,E2 -7763.761} C_VEL
LIN {X 0,Y 469.191,Z 150.92,A -85,B 0,C 180,E1 -7765.509,E2 -7765.509} C_VEL
LIN {X 0,Y 467.638,Z 143.862,A -85,B 0,C 180,E1 -7766.854,E2 -7766.854} C_VEL
LIN {X 0,Y 467.552,Z 143.873,A -85,B 0,C 180,E1 -7769.738,E2 -7769.738} C_VEL
LIN {X 0,Y 467.587,Z 143.864,A -85,B 0,C 180,E1 -7772.758,E2 -7772.758} C_VEL
LIN {X 0,Y 467.556,Z 143.868,A -85,B 0,C 180,E1 -7775.89,E2 -7775.89} C_VEL
LIN {X 0,Y 467.559,Z 143.867,A -85,B 0,C 180,E1 -7779.147,E2 -7779.147} C_VEL
LIN {X 0,Y 467.577,Z 143.869,A -85,B 0,C 180,E1 -7781.403,E2 -7781.403} C_VEL
LIN {X 0,Y 467.571,Z 143.869,A -85,B 0,C 180,E1 -7785.052,E2 -7785.052} C_VEL
LIN {X 0,Y 467.594,Z 143.864,A -85,B 0,C 180,E1 -7787.439,E2 -7787.439} C_VEL
LIN {X 0,Y 467.579,Z 143.868,A -85,B 0,C 180,E1 -7790.854,E2 -7790.854} C_VEL
LIN {X 0,Y 467.564,Z 143.87,A -85,B 0,C 180,E1 -7794.261,E2 -7794.261} C_VEL
LIN {X 0,Y 467.583,Z 143.867,A -85,B 0,C 180,E1 -7797.335,E2 -7797.335} C_VEL
LIN {X 0,Y 466.893,Z 143.954,A -85,B 0,C 180,E1 -7798.054,E2 -7798.054} C_VEL
LIN {X 0,Y 464.036,Z 144.309,A -85,B 0,C 180,E1 -7799.222,E2 -7799.222} C_VEL
LIN {X 0,Y 461.638,Z 144.609,A -85,B 0,C 180,E1 -7800.164,E2 -7800.164} C_VEL
LIN {X 0,Y 460.613,Z 144.737,A -85,B 0,C 180,E1 -7800.892,E2 -7800.892} C_VEL
LIN {X 0,Y 460.531,Z 144.745,A -85,B 0,C 180,E1 -7801.138,E2 -7801.138} C_VEL
LIN {X 0,Y 460.62,Z 144.817,A -85,B 0,C 180,E1 -7802.593,E2 -7802.593} C_VEL
LIN {X 0,Y 464.135,Z 158.984,A -85,B 0,C 180,E1 -7804.913,E2 -7804.913} C_VEL
LIN {X 0,Y 465.164,Z 163.595,A -85,B 0,C 180,E1 -7805.587,E2 -7805.587} C_VEL
LIN {X 0,Y 467.649,Z 172.479,A -85,B 0,C 180,E1 -7805.876,E2 -7805.876} C_VEL
LIN {X 0,Y 469.722,Z 181.443,A -85,B 0,C 180,E1 -7806.14,E2 -7806.14} C_VEL
LIN {X 0,Y 468.344,Z 295.383,A -85,B 0,C 180,E1 -7807.936,E2 -7807.936} C_VEL
LIN {X 0,Y 467.903,Z 331.302,A -85,B 0,C 180,E1 -7808.531,E2 -7808.531} C_VEL
LIN {X 0,Y 467.574,Z 346.518,A -85,B 0,C 180,E1 -7808.958,E2 -7808.958} C_VEL
LIN {X 0,Y 467.085,Z 360.894,A -85,B 0,C 180,E1 -7809.532,E2 -7809.532} C_VEL
LIN {X 0,Y 466.427,Z 375.404,A -85,B 0,C 180,E1 -7810.296,E2 -7810.296} C_VEL
LIN {X 0,Y 465.666,Z 388.674,A -85,B 0,C 180,E1 -7811.179,E2 -7811.179} C_VEL
LIN {X 0,Y 464.801,Z 401.153,A -85,B 0,C 180,E1 -7812.192,E2 -7812.192} C_VEL
LIN {X 0,Y 463.978,Z 413.288,A -85,B 0,C 180,E1 -7813.386,E2 -7813.386} C_VEL
LIN {X 0,Y 463.158,Z 423.669,A -85,B 0,C 180,E1 -7814.6,E2 -7814.6} C_VEL
LIN {X 0,Y 462.406,Z 433.263,A -85,B 0,C 180,E1 -7815.925,E2 -7815.925} C_VEL
LIN {X 0,Y 461.734,Z 442.175,A -85,B 0,C 180,E1 -7817.386,E2 -7817.386} C_VEL
LIN {X 0,Y 461.099,Z 450.428,A -85,B 0,C 180,E1 -7819.016,E2 -7819.016} C_VEL
LIN {X 0,Y 460.623,Z 457.673,A -85,B 0,C 180,E1 -7820.78,E2 -7820.78} C_VEL
LIN {X 0,Y 460.282,Z 463.416,A -85,B 0,C 180,E1 -7822.542,E2 -7822.542} C_VEL
LIN {X 0,Y 460.035,Z 466.808,A -85,B 0,C 180,E1 -7823.86,E2 -7823.86} C_VEL
LIN {X 0,Y 459.958,Z 470.257,A -85,B 0,C 180,E1 -7825.617,E2 -7825.617} C_VEL
LIN {X 0,Y 459.793,Z 472.543,A -85,B 0,C 180,E1 -7827.371,E2 -7827.371} C_VEL
LIN {X 0,Y 459.62,Z 473.714,A -85,B 0,C 180,E1 -7829.123,E2 -7829.123} C_VEL
LIN {X 0,Y 459.62,Z 473.73,A -85,B 0,C 180,E1 -7830.875,E2 -7830.875} C_VEL
LIN {X 0,Y 459.793,Z 472.621,A -85,B 0,C 180,E1 -7832.627,E2 -7832.627} C_VEL
LIN {X 0,Y 459.949,Z 470.402,A -85,B 0,C 180,E1 -7834.38,E2 -7834.38} C_VEL
LIN {X 0,Y 460.028,Z 467.029,A -85,B 0,C 180,E1 -7836.138,E2 -7836.138} C_VEL
LIN {X 0,Y 460.329,Z 462.387,A -85,B 0,C 180,E1 -7837.897,E2 -7837.897} C_VEL
LIN {X 0,Y 460.715,Z 456.361,A -85,B 0,C 180,E1 -7839.659,E2 -7839.659} C_VEL
LIN {X 0,Y 461.222,Z 448.777,A -85,B 0,C 180,E1 -7841.424,E2 -7841.424} C_VEL
LIN {X 0,Y 461.778,Z 441.125,A -85,B 0,C 180,E1 -7842.895,E2 -7842.895} C_VEL
LIN {X 0,Y 462.478,Z 432.434,A -85,B 0,C 180,E1 -7844.295,E2 -7844.295} C_VEL
LIN {X 0,Y 463.362,Z 420.904,A -85,B 0,C 180,E1 -7845.842,E2 -7845.842} C_VEL
LIN {X 0,Y 464.203,Z 409.828,A -85,B 0,C 180,E1 -7847.078,E2 -7847.078} C_VEL
LIN {X 0,Y 465.084,Z 397.188,A -85,B 0,C 180,E1 -7848.25,E2 -7848.25} C_VEL
LIN {X 0,Y 465.978,Z 383.803,A -85,B 0,C 180,E1 -7849.263,E2 -7849.263} C_VEL
LIN {X 0,Y 466.691,Z 369.251,A -85,B 0,C 180,E1 -7850.149,E2 -7850.149} C_VEL
LIN {X 0,Y 467.305,Z 354.534,A -85,B 0,C 180,E1 -7850.84,E2 -7850.84} C_VEL
LIN {X 0,Y 467.767,Z 340.062,A -85,B 0,C 180,E1 -7851.34,E2 -7851.34} C_VEL
LIN {X 0,Y 468.016,Z 325.924,A -85,B 0,C 180,E1 -7851.672,E2 -7851.672} C_VEL
LIN {X 0,Y 469.749,Z 182.1,A -85,B 0,C 180,E1 -7853.941,E2 -7853.941} C_VEL
LIN {X 0,Y 467.193,Z 170.706,A -85,B 0,C 180,E1 -7854.273,E2 -7854.273} C_VEL
LIN {X 0,Y 465.136,Z 163.385,A -85,B 0,C 180,E1 -7854.529,E2 -7854.529} C_VEL
LIN {X 0,Y 462.314,Z 151.494,A -85,B 0,C 180,E1 -7856.375,E2 -7856.375} C_VEL
LIN {X 0,Y 460.586,Z 144.74,A -85,B 0,C 180,E1 -7857.532,E2 -7857.532} C_VEL
LIN {X 0,Y 460.507,Z 144.749,A -85,B 0,C 180,E1 -7860.239,E2 -7860.239} C_VEL
LIN {X 0,Y 460.525,Z 144.746,A -85,B 0,C 180,E1 -7863.323,E2 -7863.323} C_VEL
LIN {X 0,Y 460.474,Z 144.749,A -85,B 0,C 180,E1 -7866.528,E2 -7866.528} C_VEL
LIN {X 0,Y 460.536,Z 144.741,A -85,B 0,C 180,E1 -7868.896,E2 -7868.896} C_VEL
LIN {X 0,Y 460.517,Z 144.744,A -85,B 0,C 180,E1 -7872.18,E2 -7872.18} C_VEL
LIN {X 0,Y 460.51,Z 144.75,A -85,B 0,C 180,E1 -7875.41,E2 -7875.41} C_VEL
LIN {X 0,Y 460.528,Z 144.74,A -85,B 0,C 180,E1 -7878.396,E2 -7878.396} C_VEL
LIN {X 0,Y 460.539,Z 144.74,A -85,B 0,C 180,E1 -7881.268,E2 -7881.268} C_VEL
LIN {X 0,Y 460.505,Z 144.744,A -85,B 0,C 180,E1 -7884.554,E2 -7884.554} C_VEL
LIN {X 0,Y 460.524,Z 144.743,A -85,B 0,C 180,E1 -7887.715,E2 -7887.715} C_VEL
LIN {X 0,Y 460.538,Z 144.735,A -85,B 0,C 180,E1 -7890.769,E2 -7890.769} C_VEL
LIN {X 0,Y 460.553,Z 144.736,A -85,B 0,C 180,E1 -7893.734,E2 -7893.734} C_VEL
LIN {X 0,Y 460.536,Z 144.738,A -85,B 0,C 180,E1 -7896.623,E2 -7896.623} C_VEL
LIN {X 0,Y 460.542,Z 144.737,A -85,B 0,C 180,E1 -7899.452,E2 -7899.452} C_VEL
LIN {X 0,Y 460.549,Z 144.734,A -85,B 0,C 180,E1 -7902.23,E2 -7902.23} C_VEL
LIN {X 0,Y 460.555,Z 144.74,A -85,B 0,C 180,E1 -7904.964,E2 -7904.964} C_VEL
LIN {X 0,Y 460.599,Z 144.725,A -85,B 0,C 180,E1 -7907.665,E2 -7907.665} C_VEL
LIN {X 0,Y 460.618,Z 144.73,A -85,B 0,C 180,E1 -7911.224,E2 -7911.224} C_VEL
LIN {X 0,Y 460.699,Z 144.708,A -85,B 0,C 180,E1 -7913.87,E2 -7913.87} C_VEL
LIN {X 0,Y 460.815,Z 144.706,A -85,B 0,C 180,E1 -7917.377,E2 -7917.377} C_VEL
LIN {X 0,Y 460.842,Z 144.693,A -85,B 0,C 180,E1 -7920,E2 -7920} C_VEL
LIN {X 0,Y 460.815,Z 144.708,A -85,B 0,C 180,E1 -7922.622,E2 -7922.622} C_VEL
LIN {X 0,Y 460.699,Z 144.715,A -85,B 0,C 180,E1 -7926.13,E2 -7926.13} C_VEL
LIN {X 0,Y 460.619,Z 144.733,A -85,B 0,C 180,E1 -7928.776,E2 -7928.776} C_VEL
LIN {X 0,Y 460.601,Z 144.726,A -85,B 0,C 180,E1 -7932.445,E2 -7932.445} C_VEL
LIN {X 0,Y 460.61,Z 144.73,A -85,B 0,C 180,E1 -7936.007,E2 -7936.007} C_VEL
LIN {X 0,Y 460.559,Z 144.728,A -85,B 0,C 180,E1 -7939.616,E2 -7939.616} C_VEL
LIN {X 0,Y 460.506,Z 144.747,A -85,B 0,C 180,E1 -7942.429,E2 -7942.429} C_VEL
LIN {X 0,Y 460.557,Z 144.734,A -85,B 0,C 180,E1 -7945.803,E2 -7945.803} C_VEL
LIN {X 0,Y 460.545,Z 144.742,A -85,B 0,C 180,E1 -7948.233,E2 -7948.233} C_VEL
LIN {X 0,Y 460.512,Z 144.743,A -85,B 0,C 180,E1 -7951.284,E2 -7951.284} C_VEL
LIN {X 0,Y 460.524,Z 144.741,A -85,B 0,C 180,E1 -7954.507,E2 -7954.507} C_VEL
LIN {X 0,Y 460.519,Z 144.743,A -85,B 0,C 180,E1 -7957.621,E2 -7957.621} C_VEL
LIN {X 0,Y 460.532,Z 144.721,A -85,B 0,C 180,E1 -7960.27,E2 -7960.27} C_VEL
LIN {X 0,Y 460.491,Z 144.746,A -85,B 0,C 180,E1 -7963.376,E2 -7963.376} C_VEL
LIN {X 0,Y 460.517,Z 144.745,A -85,B 0,C 180,E1 -7966.629,E2 -7966.629} C_VEL
LIN {X 0,Y 460.552,Z 144.743,A -85,B 0,C 180,E1 -7969.729,E2 -7969.729} C_VEL
LIN {X 0,Y 460.521,Z 144.741,A -85,B 0,C 180,E1 -7972.52,E2 -7972.52} C_VEL
LIN {X 0,Y 460.576,Z 144.859,A -85,B 0,C 180,E1 -7975.742,E2 -7975.742} C_VEL
LIN {X 0,Y 467.529,Z 167.877,A -85,B 0,C 180,E1 -7978.764,E2 -7978.764} C_VEL
LIN {X 0,Y 468.912,Z 172.622,A -85,B 0,C 180,E1 -7979.365,E2 -7979.365} C_VEL
LIN {X 0,Y 467.231,Z 198.851,A -85,B 0,C 180,E1 -7982.086,E2 -7982.086} C_VEL
LIN {X 0,Y 465.14,Z 234.309,A -85,B 0,C 180,E1 -7985.688,E2 -7985.688} C_VEL
LIN {X 0,Y 465.138,Z 235.942,A -85,B 0,C 180,E1 -7985.812,E2 -7985.812} C_VEL
LIN {X 0,Y 468.319,Z 261.427,A -85,B 0,C 180,E1 -7986.399,E2 -7986.399} C_VEL
LIN {X 0,Y 466.95,Z 383.383,A -85,B 0,C 180,E1 -7988.305,E2 -7988.305} C_VEL
LIN {X 0,Y 466.631,Z 406.062,A -85,B 0,C 180,E1 -7988.695,E2 -7988.695} C_VEL
LIN {X 0,Y 466.046,Z 421.004,A -85,B 0,C 180,E1 -7989.112,E2 -7989.112} C_VEL
LIN {X 0,Y 465.386,Z 435.261,A -85,B 0,C 180,E1 -7989.677,E2 -7989.677} C_VEL
LIN {X 0,Y 464.552,Z 449.92,A -85,B 0,C 180,E1 -7990.446,E2 -7990.446} C_VEL
LIN {X 0,Y 463.695,Z 463.28,A -85,B 0,C 180,E1 -7991.327,E2 -7991.327} C_VEL
LIN {X 0,Y 462.799,Z 476.878,A -85,B 0,C 180,E1 -7992.434,E2 -7992.434} C_VEL
LIN {X 0,Y 462.03,Z 488.769,A -85,B 0,C 180,E1 -7993.605,E2 -7993.605} C_VEL
LIN {X 0,Y 461.299,Z 500.516,A -85,B 0,C 180,E1 -7994.991,E2 -7994.991} C_VEL
LIN {X 0,Y 460.695,Z 511.469,A -85,B 0,C 180,E1 -7996.549,E2 -7996.549} C_VEL
LIN {X 0,Y 460.197,Z 519.641,A -85,B 0,C 180,E1 -7997.93,E2 -7997.93} C_VEL
LIN {X 0,Y 460.059,Z 527.136,A -85,B 0,C 180,E1 -7999.438,E2 -7999.438} C_VEL
LIN {X 0,Y 459.851,Z 534.392,A -85,B 0,C 180,E1 -8001.21,E2 -8001.21} C_VEL
LIN {X 0,Y 459.838,Z 540.107,A -85,B 0,C 180,E1 -8002.978,E2 -8002.978} C_VEL
LIN {X 0,Y 459.826,Z 544.418,A -85,B 0,C 180,E1 -8004.74,E2 -8004.74} C_VEL
LIN {X 0,Y 459.846,Z 547.442,A -85,B 0,C 180,E1 -8006.496,E2 -8006.496} C_VEL
LIN {X 0,Y 459.787,Z 549.241,A -85,B 0,C 180,E1 -8008.249,E2 -8008.249} C_VEL
LIN {X 0,Y 459.873,Z 549.864,A -85,B 0,C 180,E1 -8010.001,E2 -8010.001} C_VEL
LIN {X 0,Y 459.787,Z 549.242,A -85,B 0,C 180,E1 -8011.753,E2 -8011.753} C_VEL
LIN {X 0,Y 459.853,Z 547.444,A -85,B 0,C 180,E1 -8013.506,E2 -8013.506} C_VEL
LIN {X 0,Y 459.825,Z 544.414,A -85,B 0,C 180,E1 -8015.263,E2 -8015.263} C_VEL
LIN {X 0,Y 459.85,Z 540.096,A -85,B 0,C 180,E1 -8017.024,E2 -8017.024} C_VEL
LIN {X 0,Y 459.892,Z 534.384,A -85,B 0,C 180,E1 -8018.791,E2 -8018.791} C_VEL
LIN {X 0,Y 460.1,Z 527.131,A -85,B 0,C 180,E1 -8020.563,E2 -8020.563} C_VEL
LIN {X 0,Y 460.306,Z 519.269,A -85,B 0,C 180,E1 -8022.134,E2 -8022.134} C_VEL
LIN {X 0,Y 460.78,Z 510,A -85,B 0,C 180,E1 -8023.676,E2 -8023.676} C_VEL
LIN {X 0,Y 461.326,Z 500.491,A -85,B 0,C 180,E1 -8025.011,E2 -8025.011} C_VEL
LIN {X 0,Y 462.083,Z 488.712,A -85,B 0,C 180,E1 -8026.398,E2 -8026.398} C_VEL
LIN {X 0,Y 462.805,Z 476.825,A -85,B 0,C 180,E1 -8027.568,E2 -8027.568} C_VEL
LIN {X 0,Y 463.73,Z 463.228,A -85,B 0,C 180,E1 -8028.673,E2 -8028.673} C_VEL
LIN {X 0,Y 464.579,Z 449.859,A -85,B 0,C 180,E1 -8029.555,E2 -8029.555} C_VEL
LIN {X 0,Y 465.407,Z 435.158,A -85,B 0,C 180,E1 -8030.324,E2 -8030.324} C_VEL
LIN {X 0,Y 466.106,Z 420.088,A -85,B 0,C 180,E1 -8030.917,E2 -8030.917} C_VEL
LIN {X 0,Y 466.717,Z 404.717,A -85,B 0,C 180,E1 -8031.332,E2 -8031.332} C_VEL
LIN {X 0,Y 468.25,Z 274.944,A -85,B 0,C 180,E1 -8033.382,E2 -8033.382} C_VEL
LIN {X 0,Y 468.207,Z 259.906,A -85,B 0,C 180,E1 -8033.629,E2 -8033.629} C_VEL
LIN {X 0,Y 465.208,Z 237.089,A -85,B 0,C 180,E1 -8034.163,E2 -8034.163} C_VEL
LIN {X 0,Y 466.861,Z 213.991,A -85,B 0,C 180,E1 -8036.607,E2 -8036.607} C_VEL
LIN {X 0,Y 469.446,Z 185.844,A -85,B 0,C 180,E1 -8039.738,E2 -8039.738} C_VEL
LIN {X 0,Y 470.575,Z 175.976,A -85,B 0,C 180,E1 -8040.888,E2 -8040.888} C_VEL
LIN {X 0,Y 469.786,Z 171.889,A -85,B 0,C 180,E1 -8041.491,E2 -8041.491} C_VEL
LIN {X 0,Y 466.5,Z 160.897,A -85,B 0,C 180,E1 -8043.36,E2 -8043.36} C_VEL
LIN {X 0,Y 463.147,Z 151.593,A -85,B 0,C 180,E1 -8045.215,E2 -8045.215} C_VEL
LIN {X 0,Y 460.498,Z 144.75,A -85,B 0,C 180,E1 -8046.835,E2 -8046.835} C_VEL
LIN {X 0,Y 460.515,Z 144.749,A -85,B 0,C 180,E1 -8049.865,E2 -8049.865} C_VEL
LIN {X 0,Y 460.458,Z 144.755,A -85,B 0,C 180,E1 -8052.893,E2 -8052.893} C_VEL
LIN {X 0,Y 460.506,Z 144.75,A -85,B 0,C 180,E1 -8055.832,E2 -8055.832} C_VEL
LIN {X 0,Y 460.502,Z 144.75,A -85,B 0,C 180,E1 -8058.986,E2 -8058.986} C_VEL
LIN {X 0,Y 460.483,Z 144.752,A -85,B 0,C 180,E1 -8062.375,E2 -8062.375} C_VEL
LIN {X 0,Y 460.536,Z 144.747,A -85,B 0,C 180,E1 -8065.623,E2 -8065.623} C_VEL
LIN {X 0,Y 460.509,Z 144.785,A -85,B 0,C 180,E1 -8068.671,E2 -8068.671} C_VEL
LIN {X 0,Y 463.05,Z 152.6,A -85,B 0,C 180,E1 -8070.943,E2 -8070.943} C_VEL
LIN {X 0,Y 465.681,Z 161.733,A -85,B 0,C 180,E1 -8073.312,E2 -8073.312} C_VEL
LIN {X 0,Y 467.538,Z 170.492,A -85,B 0,C 180,E1 -8075.346,E2 -8075.346} C_VEL
LIN {X 0,Y 466.704,Z 181.321,A -85,B 0,C 180,E1 -8077.418,E2 -8077.418} C_VEL
LIN {X 0,Y 465.141,Z 199.764,A -85,B 0,C 180,E1 -8080.815,E2 -8080.815} C_VEL
LIN {X 0,Y 464.891,Z 203.95,A -85,B 0,C 180,E1 -8081.56,E2 -8081.56} C_VEL
LIN {X 0,Y 467.846,Z 216.448,A -85,B 0,C 180,E1 -8082.077,E2 -8082.077} C_VEL
LIN {X 0,Y 465.056,Z 306.059,A -85,B 0,C 180,E1 -8084.103,E2 -8084.103} C_VEL
LIN {X 0,Y 464.751,Z 322.591,A -85,B 0,C 180,E1 -8084.514,E2 -8084.514} C_VEL
LIN {X 0,Y 464.506,Z 336.085,A -85,B 0,C 180,E1 -8085.039,E2 -8085.039} C_VEL
LIN {X 0,Y 464.128,Z 349.331,A -85,B 0,C 180,E1 -8085.748,E2 -8085.748} C_VEL
LIN {X 0,Y 463.631,Z 361.345,A -85,B 0,C 180,E1 -8086.581,E2 -8086.581} C_VEL
LIN {X 0,Y 463.122,Z 373.155,A -85,B 0,C 180,E1 -8087.623,E2 -8087.623} C_VEL
LIN {X 0,Y 462.705,Z 382.242,A -85,B 0,C 180,E1 -8088.612,E2 -8088.612} C_VEL
LIN {X 0,Y 462.27,Z 390.599,A -85,B 0,C 180,E1 -8089.71,E2 -8089.71} C_VEL
LIN {X 0,Y 461.757,Z 398.745,A -85,B 0,C 180,E1 -8091.025,E2 -8091.025} C_VEL
LIN {X 0,Y 461.389,Z 404.313,A -85,B 0,C 180,E1 -8092.121,E2 -8092.121} C_VEL
LIN {X 0,Y 461.141,Z 409.693,A -85,B 0,C 180,E1 -8093.437,E2 -8093.437} C_VEL
LIN {X 0,Y 460.839,Z 413.901,A -85,B 0,C 180,E1 -8094.75,E2 -8094.75} C_VEL
LIN {X 0,Y 460.689,Z 416.094,A -85,B 0,C 180,E1 -8095.625,E2 -8095.625} C_VEL
LIN {X 0,Y 460.647,Z 417.838,A -85,B 0,C 180,E1 -8096.501,E2 -8096.501} C_VEL
LIN {X 0,Y 460.579,Z 419.121,A -85,B 0,C 180,E1 -8097.376,E2 -8097.376} C_VEL
LIN {X 0,Y 460.536,Z 419.981,A -85,B 0,C 180,E1 -8098.251,E2 -8098.251} C_VEL
LIN {X 0,Y 460.452,Z 420.451,A -85,B 0,C 180,E1 -8099.126,E2 -8099.126} C_VEL
LIN {X 0,Y 460.417,Z 420.515,A -85,B 0,C 180,E1 -8100,E2 -8100} C_VEL
LIN {X 0,Y 460.432,Z 420.129,A -85,B 0,C 180,E1 -8100.875,E2 -8100.875} C_VEL
LIN {X 0,Y 460.351,Z 419.354,A -85,B 0,C 180,E1 -8101.75,E2 -8101.75} C_VEL
LIN {X 0,Y 460.466,Z 418.158,A -85,B 0,C 180,E1 -8102.624,E2 -8102.624} C_VEL
LIN {X 0,Y 460.404,Z 415.581,A -85,B 0,C 180,E1 -8103.939,E2 -8103.939} C_VEL
LIN {X 0,Y 460.553,Z 411.973,A -85,B 0,C 180,E1 -8105.253,E2 -8105.253} C_VEL
LIN {X 0,Y 460.816,Z 407.261,A -85,B 0,C 180,E1 -8106.568,E2 -8106.568} C_VEL
LIN {X 0,Y 461.002,Z 401.331,A -85,B 0,C 180,E1 -8107.886,E2 -8107.886} C_VEL
LIN {X 0,Y 461.353,Z 393.941,A -85,B 0,C 180,E1 -8109.204,E2 -8109.204} C_VEL
LIN {X 0,Y 461.687,Z 384.746,A -85,B 0,C 180,E1 -8110.525,E2 -8110.525} C_VEL
LIN {X 0,Y 462.066,Z 374.321,A -85,B 0,C 180,E1 -8111.738,E2 -8111.738} C_VEL
LIN {X 0,Y 462.538,Z 363.705,A -85,B 0,C 180,E1 -8112.728,E2 -8112.728} C_VEL
LIN {X 0,Y 462.881,Z 352.299,A -85,B 0,C 180,E1 -8113.592,E2 -8113.592} C_VEL
LIN {X 0,Y 463.224,Z 339.98,A -85,B 0,C 180,E1 -8114.329,E2 -8114.329} C_VEL
LIN {X 0,Y 463.51,Z 326.21,A -85,B 0,C 180,E1 -8114.938,E2 -8114.938} C_VEL
LIN {X 0,Y 463.748,Z 312.609,A -85,B 0,C 180,E1 -8115.351,E2 -8115.351} C_VEL
LIN {X 0,Y 465.09,Z 213.153,A -85,B 0,C 180,E1 -8117.186,E2 -8117.186} C_VEL
LIN {X 0,Y 462.463,Z 199.059,A -85,B 0,C 180,E1 -8117.561,E2 -8117.561} C_VEL
LIN {X 0,Y 463.344,Z 179.367,A -85,B 0,C 180,E1 -8120.882,E2 -8120.882} C_VEL
LIN {X 0,Y 464.09,Z 161.747,A -85,B 0,C 180,E1 -8123.897,E2 -8123.897} C_VEL
LIN {X 0,Y 461.974,Z 150.947,A -85,B 0,C 180,E1 -8125.927,E2 -8125.927} C_VEL
LIN {X 0,Y 460.608,Z 144.737,A -85,B 0,C 180,E1 -8127.119,E2 -8127.119} C_VEL
LIN {X 0,Y 460.512,Z 144.746,A -85,B 0,C 180,E1 -8130.24,E2 -8130.24} C_VEL
LIN {X 0,Y 460.532,Z 144.747,A -85,B 0,C 180,E1 -8133.325,E2 -8133.325} C_VEL
LIN {X 0,Y 460.477,Z 144.749,A -85,B 0,C 180,E1 -8136.529,E2 -8136.529} C_VEL
LIN {X 0,Y 460.523,Z 144.738,A -85,B 0,C 180,E1 -8139.863,E2 -8139.863} C_VEL
LIN {X 0,Y 460.497,Z 144.749,A -85,B 0,C 180,E1 -8142.897,E2 -8142.897} C_VEL
LIN {X 0,Y 460.514,Z 144.744,A -85,B 0,C 180,E1 -8145.83,E2 -8145.83} C_VEL
LIN {X 0,Y 460.535,Z 144.746,A -85,B 0,C 180,E1 -8148.988,E2 -8148.988} C_VEL
LIN {X 0,Y 460.527,Z 144.748,A -85,B 0,C 180,E1 -8151.266,E2 -8151.266} C_VEL
LIN {X 0,Y 460.513,Z 144.75,A -85,B 0,C 180,E1 -8154.554,E2 -8154.554} C_VEL
LIN {X 0,Y 460.534,Z 144.744,A -85,B 0,C 180,E1 -8157.715,E2 -8157.715} C_VEL
LIN {X 0,Y 460.531,Z 144.745,A -85,B 0,C 180,E1 -8161.138,E2 -8161.138} C_VEL
LIN {X 0,Y 460.308,Z 145.152,A -85,B 0,C 180,E1 -8161.619,E2 -8161.619} C_VEL
LIN {X 0,Y 459.409,Z 146.976,A -85,B 0,C 180,E1 -8162.306,E2 -8162.306} C_VEL
LIN {X 0,Y 458.259,Z 149.796,A -85,B 0,C 180,E1 -8162.943,E2 -8162.943} C_VEL
LIN {X 0,Y 457.015,Z 154.581,A -85,B 0,C 180,E1 -8163.754,E2 -8163.754} C_VEL
LIN {X 0,Y 456.916,Z 158.441,A -85,B 0,C 180,E1 -8164.344,E2 -8164.344} C_VEL
LIN {X 0,Y 457.139,Z 159.717,A -85,B 0,C 180,E1 -8164.54,E2 -8164.54} C_VEL
LIN {X 0,Y 458.201,Z 164.189,A -85,B 0,C 180,E1 -8165.193,E2 -8165.193} C_VEL
LIN {X 0,Y 460.376,Z 170.428,A -85,B 0,C 180,E1 -8165.426,E2 -8165.426} C_VEL
LIN {X 0,Y 463.214,Z 182.282,A -85,B 0,C 180,E1 -8165.789,E2 -8165.789} C_VEL
LIN {X 0,Y 461.851,Z 294.092,A -85,B 0,C 180,E1 -8167.58,E2 -8167.58} C_VEL
LIN {X 0,Y 461.327,Z 331.817,A -85,B 0,C 180,E1 -8168.21,E2 -8168.21} C_VEL
LIN {X 0,Y 460.998,Z 346.93,A -85,B 0,C 180,E1 -8168.638,E2 -8168.638} C_VEL
LIN {X 0,Y 460.466,Z 361.544,A -85,B 0,C 180,E1 -8169.229,E2 -8169.229} C_VEL
LIN {X 0,Y 459.786,Z 375.971,A -85,B 0,C 180,E1 -8170,E2 -8170} C_VEL
LIN {X 0,Y 458.972,Z 389.247,A -85,B 0,C 180,E1 -8170.894,E2 -8170.894} C_VEL
LIN {X 0,Y 458.083,Z 401.728,A -85,B 0,C 180,E1 -8171.922,E2 -8171.922} C_VEL
LIN {X 0,Y 457.239,Z 412.838,A -85,B 0,C 180,E1 -8173.019,E2 -8173.019} C_VEL
LIN {X 0,Y 456.333,Z 424.25,A -85,B 0,C 180,E1 -8174.363,E2 -8174.363} C_VEL
LIN {X 0,Y 455.527,Z 433.846,A -85,B 0,C 180,E1 -8175.708,E2 -8175.708} C_VEL
LIN {X 0,Y 454.809,Z 442.861,A -85,B 0,C 180,E1 -8177.211,E2 -8177.211} C_VEL
LIN {X 0,Y 454.139,Z 451.013,A -85,B 0,C 180,E1 -8178.845,E2 -8178.845} C_VEL
LIN {X 0,Y 453.637,Z 458.258,A -85,B 0,C 180,E1 -8180.637,E2 -8180.637} C_VEL
LIN {X 0,Y 453.258,Z 464.001,A -85,B 0,C 180,E1 -8182.425,E2 -8182.425} C_VEL
LIN {X 0,Y 453.003,Z 467.393,A -85,B 0,C 180,E1 -8183.764,E2 -8183.764} C_VEL
LIN {X 0,Y 452.909,Z 470.841,A -85,B 0,C 180,E1 -8185.549,E2 -8185.549} C_VEL
LIN {X 0,Y 452.744,Z 473.126,A -85,B 0,C 180,E1 -8187.33,E2 -8187.33} C_VEL
LIN {X 0,Y 452.552,Z 474.299,A -85,B 0,C 180,E1 -8189.109,E2 -8189.109} C_VEL
LIN {X 0,Y 452.551,Z 474.314,A -85,B 0,C 180,E1 -8190.889,E2 -8190.889} C_VEL
LIN {X 0,Y 452.743,Z 473.204,A -85,B 0,C 180,E1 -8192.668,E2 -8192.668} C_VEL
LIN {X 0,Y 452.902,Z 470.985,A -85,B 0,C 180,E1 -8194.449,E2 -8194.449} C_VEL
LIN {X 0,Y 452.988,Z 467.612,A -85,B 0,C 180,E1 -8196.234,E2 -8196.234} C_VEL
LIN {X 0,Y 453.32,Z 462.969,A -85,B 0,C 180,E1 -8198.019,E2 -8198.019} C_VEL
LIN {X 0,Y 453.722,Z 456.944,A -85,B 0,C 180,E1 -8199.809,E2 -8199.809} C_VEL
LIN {X 0,Y 454.269,Z 449.358,A -85,B 0,C 180,E1 -8201.601,E2 -8201.601} C_VEL
LIN {X 0,Y 454.852,Z 441.957,A -85,B 0,C 180,E1 -8203.051,E2 -8203.051} C_VEL
LIN {X 0,Y 455.609,Z 433.012,A -85,B 0,C 180,E1 -8204.516,E2 -8204.516} C_VEL
LIN {X 0,Y 456.542,Z 421.478,A -85,B 0,C 180,E1 -8206.085,E2 -8206.085} C_VEL
LIN {X 0,Y 457.435,Z 410.552,A -85,B 0,C 180,E1 -8207.322,E2 -8207.322} C_VEL
LIN {X 0,Y 458.362,Z 397.754,A -85,B 0,C 180,E1 -8208.527,E2 -8208.527} C_VEL
LIN {X 0,Y 459.326,Z 384.359,A -85,B 0,C 180,E1 -8209.553,E2 -8209.553} C_VEL
LIN {X 0,Y 460.07,Z 369.798,A -85,B 0,C 180,E1 -8210.451,E2 -8210.451} C_VEL
LIN {X 0,Y 460.701,Z 355.347,A -85,B 0,C 180,E1 -8211.141,E2 -8211.141} C_VEL
LIN {X 0,Y 461.175,Z 340.161,A -85,B 0,C 180,E1 -8211.671,E2 -8211.671} C_VEL
LIN {X 0,Y 461.455,Z 324.871,A -85,B 0,C 180,E1 -8212.022,E2 -8212.022} C_VEL
LIN {X 0,Y 463.303,Z 183.167,A -85,B 0,C 180,E1 -8214.285,E2 -8214.285} C_VEL
LIN {X 0,Y 459.471,Z 167.35,A -85,B 0,C 180,E1 -8214.774,E2 -8214.774} C_VEL
LIN {X 0,Y 458.099,Z 163.786,A -85,B 0,C 180,E1 -8214.946,E2 -8214.946} C_VEL
LIN {X 0,Y 455.097,Z 151.636,A -85,B 0,C 180,E1 -8216.852,E2 -8216.852} C_VEL
LIN {X 0,Y 453.54,Z 145.618,A -85,B 0,C 180,E1 -8217.87,E2 -8217.87} C_VEL
LIN {X 0,Y 453.473,Z 145.626,A -85,B 0,C 180,E1 -8220.758,E2 -8220.758} C_VEL
LIN {X 0,Y 453.474,Z 145.625,A -85,B 0,C 180,E1 -8223.911,E2 -8223.911} C_VEL
LIN {X 0,Y 453.465,Z 145.624,A -85,B 0,C 180,E1 -8227.187,E2 -8227.187} C_VEL
LIN {X 0,Y 453.48,Z 145.61,A -85,B 0,C 180,E1 -8229.449,E2 -8229.449} C_VEL
LIN {X 0,Y 453.472,Z 145.622,A -85,B 0,C 180,E1 -8231.934,E2 -8231.934} C_VEL
LIN {X 0,Y 453.48,Z 145.626,A -85,B 0,C 180,E1 -8235.47,E2 -8235.47} C_VEL
LIN {X 0,Y 453.474,Z 145.618,A -85,B 0,C 180,E1 -8238.209,E2 -8238.209} C_VEL
LIN {X 0,Y 453.524,Z 145.615,A -85,B 0,C 180,E1 -8240.786,E2 -8240.786} C_VEL
LIN {X 0,Y 453.449,Z 145.623,A -85,B 0,C 180,E1 -8243.917,E2 -8243.917} C_VEL
LIN {X 0,Y 453.474,Z 145.625,A -85,B 0,C 180,E1 -8247.15,E2 -8247.15} C_VEL
LIN {X 0,Y 453.505,Z 145.607,A -85,B 0,C 180,E1 -8250.27,E2 -8250.27} C_VEL
LIN {X 0,Y 453.5,Z 145.619,A -85,B 0,C 180,E1 -8253.293,E2 -8253.293} C_VEL
LIN {X 0,Y 453.493,Z 145.612,A -85,B 0,C 180,E1 -8256.238,E2 -8256.238} C_VEL
LIN {X 0,Y 453.473,Z 145.621,A -85,B 0,C 180,E1 -8259.117,E2 -8259.117} C_VEL
LIN {X 0,Y 453.501,Z 145.611,A -85,B 0,C 180,E1 -8261.944,E2 -8261.944} C_VEL
LIN {X 0,Y 453.529,Z 145.619,A -85,B 0,C 180,E1 -8264.726,E2 -8264.726} C_VEL
LIN {X 0,Y 453.552,Z 145.604,A -85,B 0,C 180,E1 -8267.471,E2 -8267.471} C_VEL
LIN {X 0,Y 453.582,Z 145.608,A -85,B 0,C 180,E1 -8271.086,E2 -8271.086} C_VEL
LIN {X 0,Y 453.666,Z 145.584,A -85,B 0,C 180,E1 -8273.774,E2 -8273.774} C_VEL
LIN {X 0,Y 453.755,Z 145.585,A -85,B 0,C 180,E1 -8277.337,E2 -8277.337} C_VEL
LIN {X 0,Y 453.812,Z 145.568,A -85,B 0,C 180,E1 -8280,E2 -8280} C_VEL
LIN {X 0,Y 453.755,Z 145.588,A -85,B 0,C 180,E1 -8282.663,E2 -8282.663} C_VEL
LIN {X 0,Y 453.666,Z 145.59,A -85,B 0,C 180,E1 -8286.225,E2 -8286.225} C_VEL
LIN {X 0,Y 453.582,Z 145.607,A -85,B 0,C 180,E1 -8288.913,E2 -8288.913} C_VEL
LIN {X 0,Y 453.552,Z 145.602,A -85,B 0,C 180,E1 -8292.529,E2 -8292.529} C_VEL
LIN {X 0,Y 453.545,Z 145.612,A -85,B 0,C 180,E1 -8296.196,E2 -8296.196} C_VEL
LIN {X 0,Y 453.509,Z 145.607,A -85,B 0,C 180,E1 -8299.041,E2 -8299.041} C_VEL
LIN {X 0,Y 453.468,Z 145.621,A -85,B 0,C 180,E1 -8301.836,E2 -8301.836} C_VEL
LIN {X 0,Y 453.505,Z 145.612,A -85,B 0,C 180,E1 -8304.735,E2 -8304.735} C_VEL
LIN {X 0,Y 453.527,Z 145.617,A -85,B 0,C 180,E1 -8307.962,E2 -8307.962} C_VEL
LIN {X 0,Y 453.457,Z 145.622,A -85,B 0,C 180,E1 -8311.526,E2 -8311.526} C_VEL
LIN {X 0,Y 453.479,Z 145.619,A -85,B 0,C 180,E1 -8314.778,E2 -8314.778} C_VEL
LIN {X 0,Y 453.464,Z 145.614,A -85,B 0,C 180,E1 -8318.312,E2 -8318.312} C_VEL
LIN {X 0,Y 453.485,Z 145.598,A -85,B 0,C 180,E1 -8320.61,E2 -8320.61} C_VEL
LIN {X 0,Y 453.447,Z 145.623,A -85,B 0,C 180,E1 -8323.245,E2 -8323.245} C_VEL
LIN {X 0,Y 453.469,Z 145.626,A -85,B 0,C 180,E1 -8325.781,E2 -8325.781} C_VEL
LIN {X 0,Y 453.489,Z 145.623,A -85,B 0,C 180,E1 -8328.212,E2 -8328.212} C_VEL
LIN {X 0,Y 453.519,Z 145.614,A -85,B 0,C 180,E1 -8330.789,E2 -8330.789} C_VEL
LIN {X 0,Y 453.45,Z 145.622,A -85,B 0,C 180,E1 -8333.919,E2 -8333.919} C_VEL
LIN {X 0,Y 453.478,Z 145.676,A -85,B 0,C 180,E1 -8335.345,E2 -8335.345} C_VEL
LIN {X 0,Y 459.613,Z 165.883,A -85,B 0,C 180,E1 -8338.065,E2 -8338.065} C_VEL
LIN {X 0,Y 462.243,Z 175.182,A -85,B 0,C 180,E1 -8339.255,E2 -8339.255} C_VEL
LIN {X 0,Y 459.962,Z 207.189,A -85,B 0,C 180,E1 -8342.61,E2 -8342.61} C_VEL
LIN {X 0,Y 458.358,Z 234.628,A -85,B 0,C 180,E1 -8345.417,E2 -8345.417} C_VEL
LIN {X 0,Y 461.792,Z 262.491,A -85,B 0,C 180,E1 -8346.069,E2 -8346.069} C_VEL
LIN {X 0,Y 460.387,Z 381.143,A -85,B 0,C 180,E1 -8347.95,E2 -8347.95} C_VEL
LIN {X 0,Y 459.996,Z 405.56,A -85,B 0,C 180,E1 -8348.373,E2 -8348.373} C_VEL
LIN {X 0,Y 459.407,Z 420.594,A -85,B 0,C 180,E1 -8348.8,E2 -8348.8} C_VEL
LIN {X 0,Y 458.686,Z 434.707,A -85,B 0,C 180,E1 -8349.367,E2 -8349.367} C_VEL
LIN {X 0,Y 457.835,Z 449.357,A -85,B 0,C 180,E1 -8350.147,E2 -8350.147} C_VEL
LIN {X 0,Y 456.911,Z 462.709,A -85,B 0,C 180,E1 -8351.04,E2 -8351.04} C_VEL
LIN {X 0,Y 455.972,Z 476.301,A -85,B 0,C 180,E1 -8352.163,E2 -8352.163} C_VEL
LIN {X 0,Y 455.191,Z 487.832,A -85,B 0,C 180,E1 -8353.312,E2 -8353.312} C_VEL
LIN {X 0,Y 454.343,Z 499.93,A -85,B 0,C 180,E1 -8354.755,E2 -8354.755} C_VEL
LIN {X 0,Y 453.698,Z 510.881,A -85,B 0,C 180,E1 -8356.337,E2 -8356.337} C_VEL
LIN {X 0,Y 453.117,Z 519.731,A -85,B 0,C 180,E1 -8357.865,E2 -8357.865} C_VEL
LIN {X 0,Y 453.011,Z 526.548,A -85,B 0,C 180,E1 -8359.272,E2 -8359.272} C_VEL
LIN {X 0,Y 452.746,Z 533.8,A -85,B 0,C 180,E1 -8361.071,E2 -8361.071} C_VEL
LIN {X 0,Y 452.747,Z 539.518,A -85,B 0,C 180,E1 -8362.868,E2 -8362.868} C_VEL
LIN {X 0,Y 452.749,Z 543.832,A -85,B 0,C 180,E1 -8364.657,E2 -8364.657} C_VEL
LIN {X 0,Y 452.776,Z 546.857,A -85,B 0,C 180,E1 -8366.441,E2 -8366.441} C_VEL
LIN {X 0,Y 452.719,Z 548.657,A -85,B 0,C 180,E1 -8368.222,E2 -8368.222} C_VEL
LIN {X 0,Y 452.797,Z 549.279,A -85,B 0,C 180,E1 -8370.001,E2 -8370.001} C_VEL
LIN {X 0,Y 452.719,Z 548.658,A -85,B 0,C 180,E1 -8371.78,E2 -8371.78} C_VEL
LIN {X 0,Y 452.781,Z 546.858,A -85,B 0,C 180,E1 -8373.561,E2 -8373.561} C_VEL
LIN {X 0,Y 452.748,Z 543.827,A -85,B 0,C 180,E1 -8375.345,E2 -8375.345} C_VEL
LIN {X 0,Y 452.756,Z 539.506,A -85,B 0,C 180,E1 -8377.135,E2 -8377.135} C_VEL
LIN {X 0,Y 452.809,Z 533.793,A -85,B 0,C 180,E1 -8378.93,E2 -8378.93} C_VEL
LIN {X 0,Y 453.035,Z 526.539,A -85,B 0,C 180,E1 -8380.73,E2 -8380.73} C_VEL
LIN {X 0,Y 453.31,Z 518.353,A -85,B 0,C 180,E1 -8382.384,E2 -8382.384} C_VEL
LIN {X 0,Y 453.769,Z 509.407,A -85,B 0,C 180,E1 -8383.891,E2 -8383.891} C_VEL
LIN {X 0,Y 454.368,Z 499.901,A -85,B 0,C 180,E1 -8385.246,E2 -8385.246} C_VEL
LIN {X 0,Y 455.183,Z 487.84,A -85,B 0,C 180,E1 -8386.684,E2 -8386.684} C_VEL
LIN {X 0,Y 455.992,Z 476.244,A -85,B 0,C 180,E1 -8387.839,E2 -8387.839} C_VEL
LIN {X 0,Y 456.95,Z 462.65,A -85,B 0,C 180,E1 -8388.961,E2 -8388.961} C_VEL
LIN {X 0,Y 457.827,Z 449.285,A -85,B 0,C 180,E1 -8389.856,E2 -8389.856} C_VEL
LIN {X 0,Y 458.753,Z 434.598,A -85,B 0,C 180,E1 -8390.632,E2 -8390.632} C_VEL
LIN {X 0,Y 459.447,Z 419.56,A -85,B 0,C 180,E1 -8391.234,E2 -8391.234} C_VEL
LIN {X 0,Y 460.082,Z 404.199,A -85,B 0,C 180,E1 -8391.655,E2 -8391.655} C_VEL
LIN {X 0,Y 461.53,Z 289.718,A -85,B 0,C 180,E1 -8393.491,E2 -8393.491} C_VEL
LIN {X 0,Y 461.7,Z 260.866,A -85,B 0,C 180,E1 -8393.959,E2 -8393.959} C_VEL
LIN {X 0,Y 458.918,Z 239.407,A -85,B 0,C 180,E1 -8394.468,E2 -8394.468} C_VEL
LIN {X 0,Y 458.611,Z 236.789,A -85,B 0,C 180,E1 -8394.562,E2 -8394.562} C_VEL
LIN {X 0,Y 460.65,Z 211.074,A -85,B 0,C 180,E1 -8397.365,E2 -8397.365} C_VEL
LIN {X 0,Y 463.305,Z 185.61,A -85,B 0,C 180,E1 -8400.291,E2 -8400.291} C_VEL
LIN {X 0,Y 464.161,Z 177.43,A -85,B 0,C 180,E1 -8401.288,E2 -8401.288} C_VEL
LIN {X 0,Y 461.668,Z 168.185,A -85,B 0,C 180,E1 -8402.83,E2 -8402.83} C_VEL
LIN {X 0,Y 458.744,Z 159.323,A -85,B 0,C 180,E1 -8404.531,E2 -8404.531} C_VEL
LIN {X 0,Y 455.767,Z 151.619,A -85,B 0,C 180,E1 -8406.282,E2 -8406.282} C_VEL
LIN {X 0,Y 453.461,Z 145.628,A -85,B 0,C 180,E1 -8407.89,E2 -8407.89} C_VEL
LIN {X 0,Y 453.473,Z 145.625,A -85,B 0,C 180,E1 -8410.612,E2 -8410.612} C_VEL
LIN {X 0,Y 453.483,Z 145.623,A -85,B 0,C 180,E1 -8414.529,E2 -8414.529} C_VEL
LIN {X 0,Y 453.433,Z 145.629,A -85,B 0,C 180,E1 -8418.072,E2 -8418.072} C_VEL
LIN {X 0,Y 453.426,Z 145.631,A -85,B 0,C 180,E1 -8420.805,E2 -8420.805} C_VEL
LIN {X 0,Y 453.443,Z 145.629,A -85,B 0,C 180,E1 -8423.916,E2 -8423.916} C_VEL
LIN {X 0,Y 453.482,Z 145.626,A -85,B 0,C 180,E1 -8426.814,E2 -8426.814} C_VEL
LIN {X 0,Y 453.483,Z 145.733,A -85,B 0,C 180,E1 -8427.645,E2 -8427.645} C_VEL
LIN {X 0,Y 456.112,Z 153.406,A -85,B 0,C 180,E1 -8430.093,E2 -8430.093} C_VEL
LIN {X 0,Y 458.855,Z 162.751,A -85,B 0,C 180,E1 -8432.668,E2 -8432.668} C_VEL
LIN {X 0,Y 460.949,Z 172.215,A -85,B 0,C 180,E1 -8434.97,E2 -8434.97} C_VEL
LIN {X 0,Y 460.96,Z 175.686,A -85,B 0,C 180,E1 -8435.691,E2 -8435.691} C_VEL
LIN {X 0,Y 459.413,Z 191.542,A -85,B 0,C 180,E1 -8438.722,E2 -8438.722} C_VEL
LIN {X 0,Y 458.351,Z 204.584,A -85,B 0,C 180,E1 -8441.129,E2 -8441.129} C_VEL
LIN {X 0,Y 461.522,Z 217.621,A -85,B 0,C 180,E1 -8441.7,E2 -8441.7} C_VEL
LIN {X 0,Y 458.431,Z 307.698,A -85,B 0,C 180,E1 -8443.81,E2 -8443.81} C_VEL
LIN {X 0,Y 458.151,Z 324.624,A -85,B 0,C 180,E1 -8444.257,E2 -8444.257} C_VEL
LIN {X 0,Y 457.863,Z 337.086,A -85,B 0,C 180,E1 -8444.76,E2 -8444.76} C_VEL
LIN {X 0,Y 457.399,Z 350.951,A -85,B 0,C 180,E1 -8445.519,E2 -8445.519} C_VEL
LIN {X 0,Y 456.882,Z 362.719,A -85,B 0,C 180,E1 -8446.359,E2 -8446.359} C_VEL
LIN {X 0,Y 456.325,Z 374.644,A -85,B 0,C 180,E1 -8447.435,E2 -8447.435} C_VEL
LIN {X 0,Y 455.884,Z 383.64,A -85,B 0,C 180,E1 -8448.439,E2 -8448.439} C_VEL
LIN {X 0,Y 455.331,Z 393.38,A -85,B 0,C 180,E1 -8449.776,E2 -8449.776} C_VEL
LIN {X 0,Y 454.838,Z 401.211,A -85,B 0,C 180,E1 -8451.111,E2 -8451.111} C_VEL
LIN {X 0,Y 454.411,Z 407.486,A -85,B 0,C 180,E1 -8452.446,E2 -8452.446} C_VEL
LIN {X 0,Y 454.054,Z 412.443,A -85,B 0,C 180,E1 -8453.78,E2 -8453.78} C_VEL
LIN {X 0,Y 453.84,Z 416.23,A -85,B 0,C 180,E1 -8455.114,E2 -8455.114} C_VEL
LIN {X 0,Y 453.675,Z 418.96,A -85,B 0,C 180,E1 -8456.447,E2 -8456.447} C_VEL
LIN {X 0,Y 453.584,Z 420.216,A -85,B 0,C 180,E1 -8457.336,E2 -8457.336} C_VEL
LIN {X 0,Y 453.521,Z 421.054,A -85,B 0,C 180,E1 -8458.224,E2 -8458.224} C_VEL
LIN {X 0,Y 453.432,Z 421.502,A -85,B 0,C 180,E1 -8459.112,E2 -8459.112} C_VEL
LIN {X 0,Y 453.395,Z 421.54,A -85,B 0,C 180,E1 -8460,E2 -8460} C_VEL
LIN {X 0,Y 453.41,Z 421.124,A -85,B 0,C 180,E1 -8460.888,E2 -8460.888} C_VEL
LIN {X 0,Y 453.328,Z 420.321,A -85,B 0,C 180,E1 -8461.777,E2 -8461.777} C_VEL
LIN {X 0,Y 453.444,Z 419.094,A -85,B 0,C 180,E1 -8462.665,E2 -8462.665} C_VEL
LIN {X 0,Y 453.383,Z 416.465,A -85,B 0,C 180,E1 -8464,E2 -8464} C_VEL
LIN {X 0,Y 453.548,Z 412.799,A -85,B 0,C 180,E1 -8465.335,E2 -8465.335} C_VEL
LIN {X 0,Y 453.846,Z 407.525,A -85,B 0,C 180,E1 -8466.789,E2 -8466.789} C_VEL
LIN {X 0,Y 454.072,Z 400.874,A -85,B 0,C 180,E1 -8468.231,E2 -8468.231} C_VEL
LIN {X 0,Y 454.427,Z 393.115,A -85,B 0,C 180,E1 -8469.57,E2 -8469.57} C_VEL
LIN {X 0,Y 454.785,Z 383.529,A -85,B 0,C 180,E1 -8470.912,E2 -8470.912} C_VEL
LIN {X 0,Y 455.2,Z 373.596,A -85,B 0,C 180,E1 -8472.031,E2 -8472.031} C_VEL
LIN {X 0,Y 455.678,Z 362.645,A -85,B 0,C 180,E1 -8473.036,E2 -8473.036} C_VEL
LIN {X 0,Y 456.029,Z 350.489,A -85,B 0,C 180,E1 -8473.933,E2 -8473.933} C_VEL
LIN {X 0,Y 456.421,Z 337.648,A -85,B 0,C 180,E1 -8474.661,E2 -8474.661} C_VEL
LIN {X 0,Y 456.655,Z 325.894,A -85,B 0,C 180,E1 -8475.167,E2 -8475.167} C_VEL
LIN {X 0,Y 456.868,Z 312.984,A -85,B 0,C 180,E1 -8475.56,E2 -8475.56} C_VEL
LIN {X 0,Y 458.328,Z 214.183,A -85,B 0,C 180,E1 -8477.424,E2 -8477.424} C_VEL
LIN {X 0,Y 455.548,Z 199.309,A -85,B 0,C 180,E1 -8477.831,E2 -8477.831} C_VEL
LIN {X 0,Y 456.495,Z 179.48,A -85,B 0,C 180,E1 -8481.211,E2 -8481.211} C_VEL
LIN {X 0,Y 457.184,Z 164.5,A -85,B 0,C 180,E1 -8483.799,E2 -8483.799} C_VEL
LIN {X 0,Y 456.748,Z 160.416,A -85,B 0,C 180,E1 -8484.548,E2 -8484.548} C_VEL
LIN {X 0,Y 453.521,Z 145.62,A -85,B 0,C 180,E1 -8487.422,E2 -8487.422} C_VEL
LIN {X 0,Y 453.48,Z 145.622,A -85,B 0,C 180,E1 -8490.759,E2 -8490.759} C_VEL
LIN {X 0,Y 453.481,Z 145.622,A -85,B 0,C 180,E1 -8493.913,E2 -8493.913} C_VEL
LIN {X 0,Y 453.454,Z 145.629,A -85,B 0,C 180,E1 -8497.19,E2 -8497.19} C_VEL
LIN {X 0,Y 453.498,Z 145.613,A -85,B 0,C 180,E1 -8500.609,E2 -8500.609} C_VEL
LIN {X 0,Y 453.465,Z 145.618,A -85,B 0,C 180,E1 -8504.221,E2 -8504.221} C_VEL
LIN {X 0,Y 453.468,Z 145.622,A -85,B 0,C 180,E1 -8507.005,E2 -8507.005} C_VEL
LIN {X 0,Y 453.499,Z 145.617,A -85,B 0,C 180,E1 -8509.409,E2 -8509.409} C_VEL
LIN {X 0,Y 453.454,Z 145.626,A -85,B 0,C 180,E1 -8512.227,E2 -8512.227} C_VEL
LIN {X 0,Y 453.487,Z 145.624,A -85,B 0,C 180,E1 -8515.223,E2 -8515.223} C_VEL
LIN {X 0,Y 453.47,Z 145.625,A -85,B 0,C 180,E1 -8518.474,E2 -8518.474} C_VEL
LIN {X 0,Y 453.536,Z 145.618,A -85,B 0,C 180,E1 -8522.04,E2 -8522.04} C_VEL
LIN {X 0,Y 453.56,Z 145.736,A -85,B 0,C 180,E1 -8522.235,E2 -8522.235} C_VEL
LIN {X 0,Y 457.075,Z 159.447,A -85,B 0,C 180,E1 -8524.498,E2 -8524.498} C_VEL
LIN {X 0,Y 457.139,Z 159.717,A -85,B 0,C 180,E1 -8524.54,E2 -8524.54} C_VEL
LIN {X 0,Y 457.708,Z 162.555,A -85,B 0,C 180,E1 -8524.867,E2 -8524.867} C_VEL
LIN {X 0,Y 458.184,Z 165.954,A -85,B 0,C 180,E1 -8525.104,E2 -8525.104} C_VEL
LIN {X 0,Y 458.511,Z 171.64,A -85,B 0,C 180,E1 -8525.324,E2 -8525.324} C_VEL
LIN {X 0,Y 458.047,Z 177.797,A -85,B 0,C 180,E1 -8525.415,E2 -8525.415} C_VEL
LIN {X 0,Y 457.413,Z 181.998,A -85,B 0,C 180,E1 -8525.45,E2 -8525.45} C_VEL
LIN {X 0,Y 456.787,Z 190.412,A -85,B 0,C 180,E1 -8525.557,E2 -8525.557} C_VEL
LIN {X 0,Y 454.766,Z 331.12,A -85,B 0,C 180,E1 -8527.852,E2 -8527.852} C_VEL
LIN {X 0,Y 454.481,Z 345.974,A -85,B 0,C 180,E1 -8528.264,E2 -8528.264} C_VEL
LIN {X 0,Y 454.005,Z 358.82,A -85,B 0,C 180,E1 -8528.761,E2 -8528.761} C_VEL
LIN {X 0,Y 453.369,Z 372.732,A -85,B 0,C 180,E1 -8529.467,E2 -8529.467} C_VEL
LIN {X 0,Y 452.478,Z 386.78,A -85,B 0,C 180,E1 -8530.373,E2 -8530.373} C_VEL
LIN {X 0,Y 451.546,Z 399.567,A -85,B 0,C 180,E1 -8531.392,E2 -8531.392} C_VEL
LIN {X 0,Y 450.608,Z 411.895,A -85,B 0,C 180,E1 -8532.589,E2 -8532.589} C_VEL
LIN {X 0,Y 449.641,Z 423.111,A -85,B 0,C 180,E1 -8533.892,E2 -8533.892} C_VEL
LIN {X 0,Y 448.799,Z 432.973,A -85,B 0,C 180,E1 -8535.257,E2 -8535.257} C_VEL
LIN {X 0,Y 447.996,Z 442.048,A -85,B 0,C 180,E1 -8536.753,E2 -8536.753} C_VEL
LIN {X 0,Y 447.287,Z 450.571,A -85,B 0,C 180,E1 -8538.442,E2 -8538.442} C_VEL
LIN {X 0,Y 446.735,Z 457.167,A -85,B 0,C 180,E1 -8540.034,E2 -8540.034} C_VEL
LIN {X 0,Y 446.312,Z 463.262,A -85,B 0,C 180,E1 -8541.851,E2 -8541.851} C_VEL
LIN {X 0,Y 445.969,Z 467.978,A -85,B 0,C 180,E1 -8543.666,E2 -8543.666} C_VEL
LIN {X 0,Y 445.863,Z 471.426,A -85,B 0,C 180,E1 -8545.479,E2 -8545.479} C_VEL
LIN {X 0,Y 445.696,Z 473.71,A -85,B 0,C 180,E1 -8547.287,E2 -8547.287} C_VEL
LIN {X 0,Y 445.486,Z 474.883,A -85,B 0,C 180,E1 -8549.095,E2 -8549.095} C_VEL
LIN {X 0,Y 445.485,Z 474.898,A -85,B 0,C 180,E1 -8550.903,E2 -8550.903} C_VEL
LIN {X 0,Y 445.695,Z 473.786,A -85,B 0,C 180,E1 -8552.71,E2 -8552.71} C_VEL
LIN {X 0,Y 445.854,Z 471.568,A -85,B 0,C 180,E1 -8554.519,E2 -8554.519} C_VEL
LIN {X 0,Y 445.951,Z 468.195,A -85,B 0,C 180,E1 -8556.332,E2 -8556.332} C_VEL
LIN {X 0,Y 446.292,Z 463.553,A -85,B 0,C 180,E1 -8558.147,E2 -8558.147} C_VEL
LIN {X 0,Y 446.723,Z 457.527,A -85,B 0,C 180,E1 -8559.964,E2 -8559.964} C_VEL
LIN {X 0,Y 447.323,Z 449.938,A -85,B 0,C 180,E1 -8561.784,E2 -8561.784} C_VEL
LIN {X 0,Y 448.059,Z 441.313,A -85,B 0,C 180,E1 -8563.468,E2 -8563.468} C_VEL
LIN {X 0,Y 448.9,Z 432.051,A -85,B 0,C 180,E1 -8564.969,E2 -8564.969} C_VEL
LIN {X 0,Y 449.745,Z 422.051,A -85,B 0,C 180,E1 -8566.335,E2 -8566.335} C_VEL
LIN {X 0,Y 450.741,Z 409.836,A -85,B 0,C 180,E1 -8567.722,E2 -8567.722} C_VEL
LIN {X 0,Y 451.694,Z 398.043,A -85,B 0,C 180,E1 -8568.834,E2 -8568.834} C_VEL
LIN {X 0,Y 452.658,Z 384.918,A -85,B 0,C 180,E1 -8569.853,E2 -8569.853} C_VEL
LIN {X 0,Y 453.458,Z 370.345,A -85,B 0,C 180,E1 -8570.763,E2 -8570.763} C_VEL
LIN {X 0,Y 454.105,Z 355.745,A -85,B 0,C 180,E1 -8571.469,E2 -8571.469} C_VEL
LIN {X 0,Y 454.618,Z 340.663,A -85,B 0,C 180,E1 -8572,E2 -8572} C_VEL
LIN {X 0,Y 454.882,Z 327.119,A -85,B 0,C 180,E1 -8572.325,E2 -8572.325} C_VEL
LIN {X 0,Y 456.851,Z 183.778,A -85,B 0,C 180,E1 -8574.648,E2 -8574.648} C_VEL
LIN {X 0,Y 453.245,Z 169.702,A -85,B 0,C 180,E1 -8575.104,E2 -8575.104} C_VEL
LIN {X 0,Y 451.063,Z 164.384,A -85,B 0,C 180,E1 -8575.352,E2 -8575.352} C_VEL
LIN {X 0,Y 447.969,Z 151.943,A -85,B 0,C 180,E1 -8577.314,E2 -8577.314} C_VEL
LIN {X 0,Y 446.467,Z 146.498,A -85,B 0,C 180,E1 -8578.246,E2 -8578.246} C_VEL
LIN {X 0,Y 446.416,Z 146.496,A -85,B 0,C 180,E1 -8581.774,E2 -8581.774} C_VEL
LIN {X 0,Y 446.426,Z 146.501,A -85,B 0,C 180,E1 -8584.522,E2 -8584.522} C_VEL
LIN {X 0,Y 446.424,Z 146.5,A -85,B 0,C 180,E1 -8588.08,E2 -8588.08} C_VEL
LIN {X 0,Y 446.421,Z 146.487,A -85,B 0,C 180,E1 -8590.916,E2 -8590.916} C_VEL
LIN {X 0,Y 446.416,Z 146.497,A -85,B 0,C 180,E1 -8593.842,E2 -8593.842} C_VEL
LIN {X 0,Y 446.392,Z 146.503,A -85,B 0,C 180,E1 -8596.402,E2 -8596.402} C_VEL
LIN {X 0,Y 446.461,Z 146.494,A -85,B 0,C 180,E1 -8599.804,E2 -8599.804} C_VEL
LIN {X 0,Y 446.426,Z 146.497,A -85,B 0,C 180,E1 -8602.123,E2 -8602.123} C_VEL
LIN {X 0,Y 446.422,Z 146.496,A -85,B 0,C 180,E1 -8605.476,E2 -8605.476} C_VEL
LIN {X 0,Y 446.425,Z 146.501,A -85,B 0,C 180,E1 -8608.7,E2 -8608.7} C_VEL
LIN {X 0,Y 446.475,Z 146.492,A -85,B 0,C 180,E1 -8611.821,E2 -8611.821} C_VEL
LIN {X 0,Y 446.447,Z 146.492,A -85,B 0,C 180,E1 -8614.847,E2 -8614.847} C_VEL
LIN {X 0,Y 446.438,Z 146.497,A -85,B 0,C 180,E1 -8618.244,E2 -8618.244} C_VEL
LIN {X 0,Y 446.447,Z 146.49,A -85,B 0,C 180,E1 -8621.649,E2 -8621.649} C_VEL
LIN {X 0,Y 446.497,Z 146.492,A -85,B 0,C 180,E1 -8624.479,E2 -8624.479} C_VEL
LIN {X 0,Y 446.504,Z 146.482,A -85,B 0,C 180,E1 -8627.383,E2 -8627.383} C_VEL
LIN {X 0,Y 446.528,Z 146.488,A -85,B 0,C 180,E1 -8630.944,E2 -8630.944} C_VEL
LIN {X 0,Y 446.636,Z 146.46,A -85,B 0,C 180,E1 -8633.676,E2 -8633.676} C_VEL
LIN {X 0,Y 446.699,Z 146.464,A -85,B 0,C 180,E1 -8637.295,E2 -8637.295} C_VEL
LIN {X 0,Y 446.783,Z 146.443,A -85,B 0,C 180,E1 -8640,E2 -8640} C_VEL
LIN {X 0,Y 446.699,Z 146.468,A -85,B 0,C 180,E1 -8642.705,E2 -8642.705} C_VEL
LIN {X 0,Y 446.635,Z 146.464,A -85,B 0,C 180,E1 -8646.324,E2 -8646.324} C_VEL
LIN {X 0,Y 446.528,Z 146.485,A -85,B 0,C 180,E1 -8649.055,E2 -8649.055} C_VEL
LIN {X 0,Y 446.51,Z 146.477,A -85,B 0,C 180,E1 -8652.73,E2 -8652.73} C_VEL
LIN {X 0,Y 446.508,Z 146.49,A -85,B 0,C 180,E1 -8656.238,E2 -8656.238} C_VEL
LIN {X 0,Y 446.458,Z 146.484,A -85,B 0,C 180,E1 -8659.304,E2 -8659.304} C_VEL
LIN {X 0,Y 446.411,Z 146.504,A -85,B 0,C 180,E1 -8662.2,E2 -8662.2} C_VEL
LIN {X 0,Y 446.448,Z 146.49,A -85,B 0,C 180,E1 -8665.153,E2 -8665.153} C_VEL
LIN {X 0,Y 446.474,Z 146.495,A -85,B 0,C 180,E1 -8668.179,E2 -8668.179} C_VEL
LIN {X 0,Y 446.41,Z 146.502,A -85,B 0,C 180,E1 -8671.776,E2 -8671.776} C_VEL
LIN {X 0,Y 446.421,Z 146.497,A -85,B 0,C 180,E1 -8674.524,E2 -8674.524} C_VEL
LIN {X 0,Y 446.421,Z 146.495,A -85,B 0,C 180,E1 -8678.083,E2 -8678.083} C_VEL
LIN {X 0,Y 446.418,Z 146.479,A -85,B 0,C 180,E1 -8680.919,E2 -8680.919} C_VEL
LIN {X 0,Y 446.393,Z 146.506,A -85,B 0,C 180,E1 -8683.847,E2 -8683.847} C_VEL
LIN {X 0,Y 446.439,Z 146.501,A -85,B 0,C 180,E1 -8686.398,E2 -8686.398} C_VEL
LIN {X 0,Y 446.46,Z 146.498,A -85,B 0,C 180,E1 -8689.806,E2 -8689.806} C_VEL
LIN {X 0,Y 446.425,Z 146.499,A -85,B 0,C 180,E1 -8692.125,E2 -8692.125} C_VEL
LIN {X 0,Y 446.426,Z 146.508,A -85,B 0,C 180,E1 -8694.947,E2 -8694.947} C_VEL
LIN {X 0,Y 452.579,Z 166.809,A -85,B 0,C 180,E1 -8697.728,E2 -8697.728} C_VEL
LIN {X 0,Y 455.5,Z 176.878,A -85,B 0,C 180,E1 -8699.048,E2 -8699.048} C_VEL
LIN {X 0,Y 453.171,Z 208.342,A -85,B 0,C 180,E1 -8702.4,E2 -8702.4} C_VEL
LIN {X 0,Y 451.651,Z 233.509,A -85,B 0,C 180,E1 -8705.016,E2 -8705.016} C_VEL
LIN {X 0,Y 455.294,Z 263.119,A -85,B 0,C 180,E1 -8705.724,E2 -8705.724} C_VEL
LIN {X 0,Y 453.756,Z 384.297,A -85,B 0,C 180,E1 -8707.671,E2 -8707.671} C_VEL
LIN {X 0,Y 453.387,Z 405.058,A -85,B 0,C 180,E1 -8708.041,E2 -8708.041} C_VEL
LIN {X 0,Y 452.785,Z 420.132,A -85,B 0,C 180,E1 -8708.477,E2 -8708.477} C_VEL
LIN {X 0,Y 451.998,Z 434.154,A -85,B 0,C 180,E1 -8709.047,E2 -8709.047} C_VEL
LIN {X 0,Y 451.123,Z 448.794,A -85,B 0,C 180,E1 -8709.839,E2 -8709.839} C_VEL
LIN {X 0,Y 450.121,Z 462.136,A -85,B 0,C 180,E1 -8710.743,E2 -8710.743} C_VEL
LIN {X 0,Y 449.123,Z 475.721,A -85,B 0,C 180,E1 -8711.881,E2 -8711.881} C_VEL
LIN {X 0,Y 448.38,Z 486.46,A -85,B 0,C 180,E1 -8712.965,E2 -8712.965} C_VEL
LIN {X 0,Y 447.548,Z 497.564,A -85,B 0,C 180,E1 -8714.285,E2 -8714.285} C_VEL
LIN {X 0,Y 446.832,Z 507.334,A -85,B 0,C 180,E1 -8715.658,E2 -8715.658} C_VEL
LIN {X 0,Y 446.297,Z 516.934,A -85,B 0,C 180,E1 -8717.265,E2 -8717.265} C_VEL
LIN {X 0,Y 445.971,Z 524.926,A -85,B 0,C 180,E1 -8718.871,E2 -8718.871} C_VEL
LIN {X 0,Y 445.694,Z 531.556,A -85,B 0,C 180,E1 -8720.471,E2 -8720.471} C_VEL
LIN {X 0,Y 445.658,Z 537.653,A -85,B 0,C 180,E1 -8722.298,E2 -8722.298} C_VEL
LIN {X 0,Y 445.663,Z 541.255,A -85,B 0,C 180,E1 -8723.664,E2 -8723.664} C_VEL
LIN {X 0,Y 445.681,Z 544.914,A -85,B 0,C 180,E1 -8725.479,E2 -8725.479} C_VEL
LIN {X 0,Y 445.738,Z 547.327,A -85,B 0,C 180,E1 -8727.29,E2 -8727.29} C_VEL
LIN {X 0,Y 445.706,Z 548.535,A -85,B 0,C 180,E1 -8729.098,E2 -8729.098} C_VEL
LIN {X 0,Y 445.683,Z 548.533,A -85,B 0,C 180,E1 -8730.905,E2 -8730.905} C_VEL
LIN {X 0,Y 445.74,Z 547.328,A -85,B 0,C 180,E1 -8732.712,E2 -8732.712} C_VEL
LIN {X 0,Y 445.665,Z 544.911,A -85,B 0,C 180,E1 -8734.523,E2 -8734.523} C_VEL
LIN {X 0,Y 445.665,Z 541.244,A -85,B 0,C 180,E1 -8736.339,E2 -8736.339} C_VEL
LIN {X 0,Y 445.693,Z 536.241,A -85,B 0,C 180,E1 -8738.16,E2 -8738.16} C_VEL
LIN {X 0,Y 445.784,Z 529.776,A -85,B 0,C 180,E1 -8739.988,E2 -8739.988} C_VEL
LIN {X 0,Y 446.062,Z 522.807,A -85,B 0,C 180,E1 -8741.59,E2 -8741.59} C_VEL
LIN {X 0,Y 446.441,Z 514.391,A -85,B 0,C 180,E1 -8743.196,E2 -8743.196} C_VEL
LIN {X 0,Y 447.058,Z 504.264,A -85,B 0,C 180,E1 -8744.802,E2 -8744.802} C_VEL
LIN {X 0,Y 447.78,Z 493.908,A -85,B 0,C 180,E1 -8746.177,E2 -8746.177} C_VEL
